(* CODESYS project TcDynCollections.library
   Company: FisoThemes
   DefaultNamespace: TcDynCollections
   Version: 0.3.1.0
   DocFormat: reStructuredText
   Placeholder: TwinCat Dynamic Collections
   Author: Goodwill Mzumala
   Description: A library for handling collections of data dynamically.
   Title: TwinCat Dynamic Collections

Project tree, tasks and I/O mapping:
  libraries: Tc2_Standard, * (Beckhoff Automation GmbH); Tc2_System, * (Beckhoff Automation GmbH); Tc2_Utilities, 3.3.38.0 (Beckhoff Automation GmbH); Tc3_Module, * (Beckhoff Automation GmbH)
  DUTs/
    Aliases/
      data type T_BST_Node
      data type T_BST_Traversal
      data type T_Capacity
      data type T_Error
      data type T_Generic
      data type T_Generic_Ex
      data type T_Hash_Code
      data type T_Query_Interface
      data type T_Type
    Enums/
      data type E_BINARY_SEARCH_TREE_TRAVERSAL
    Interfaces/
      interface I_Binary_Search_Tree: _Type, Balance, Find, Insert, Remove, Traverse
      interface I_Collection: _Count, _Error_Status, _Is_Empty, Clear
      interface I_Deque: Back, Dequeue_At_Back, Dequeue_At_Front, Dequeue_Void_At_Back, Dequeue_Void_At_Front, Enqueue_At_Back, Enqueue_At_Front, Front, Peek, Reverse
      interface I_Generic_Binary_Search_Tree: Find_Generic, Insert_Generic
      interface I_Generic_Collection
      interface I_Generic_List: Get_Generic, Insert_Generic
      interface I_List: Add_Back, Add_Front, Contains, Find, Get, Get_First, Get_Last, Get_Value_As_String, Insert, Remove, Remove_At, Remove_Last, Resize, Reverse, Set
      interface I_Map: _Keys, _Values, Get, Insert, Remove, Update
      interface I_Queue: Dequeue, Dequeue_Void, Enqueue, Enqueue_At_Front, Peek, Reverse
      interface I_Read_Only_List: Clear, Contains, Find, Get, Get_First, Get_Last, Get_Value_As_String
      interface I_Stack: Peek, Pop, Pop_Void, Push, Reverse, Top
      interface I_Tree_Map: _Traversal, Balance
      interface I_Write_Only_List: _Count, _Is_Empty, Add_Back, Add_Front, Clear, Insert, Remove, Remove_At, Remove_Last, Resize, Reverse, Set
    Structs/
      data type ST_BINARY_SEARCH_TREE_NODE
      data type ST_ERROR
      data type ST_GENERIC
      data type ST_HASH_MAP_ENTRY
      data type ST_LIST_NODE
      data type ST_TREE_MAP_ENTRY_NODE
  GVLs/
    global variables GVL_CmpErrors
  POUs/
    Examples/
      program P_Example_Array_List [ST]: Scrub
      program P_Example_Binary_Search_Tree [ST]
      program P_Example_List [ST]: Scrub
      program P_Example_Queue [ST]
      program P_Example_Stack [ST]
      program P_Example_Tree_Map [ST]: Scrub
    Function Blocks/
      Helpers/
        function block FB_Helper_BST_Balancer [ST]
        function block FB_Helper_Tree_Map_Balancer [ST]
      function block FB_Array_List [ST]: EmptyListException, LessThanZeroException, MemCmpErrExpection, OutOfBoundsException, TypeMismatchException, CopyValueTo, DecrementCount, Free_Value, GetValueAsString, IncrementCount, Internal_Add_Back, Internal_Add_Front, Internal_Set, Malloc_Array, Malloc_Value, SetValue, _Is_Empty, Add_Back, Add_Front, Clear, Contains, FB_exit, FB_init, Find, Get, Get_First, Get_Generic, Get_Last, Get_Value_As_String, Insert, Insert_Generic, Remove, Remove_At, Remove_Last, Resize, Reverse, Set
      function block FB_Binary_Search_Tree [ST]: InvalidTypeException, Balance_Ready, Compare, Internal_Find, Internal_Insert, Internal_Remove, Is_Balanced, Malloc_Node, _Type, Balance, Clear, FB_exit, FB_init, Find, Find_Generic, Insert, Insert_Generic, Remove, Traverse
      function block FB_Collection [ST]: ClearException, EmptyListException, FailedInsertionException, NullReferenceException, OutOfBoundsException, RaiseException, ValueFoundException, ValueNotFoundException, ClearValue, CopyValueTo, DecrementCount, IncrementCount, _Count, _Error_Status, _Is_Empty, Clear
      function block FB_Hash_Map [ST]: Populate_Bucket_List, FB_init, Get, Insert, Remove, Remove_Void, Update
      function block FB_List [ST]: EmptyListException, MemCmpErrExpection, OutOfBoundsException, TypeMismatchException, CopyValueTo, DecrementCount, Free_Node, GetValueAsString, IncrementCount, Iterate, Malloc_Node, SetValue, _Is_Empty, Add_Back, Add_Front, Clear, Contains, FB_exit, FB_init, Find, Get, Get_First, Get_Generic, Get_Last, Get_Value_As_String, Insert, Insert_Generic, Remove, Remove_At, Remove_Last, Resize, Reverse, Set
      function block FB_Queue [ST]: NullReferenceException, _Count, _Error_Status, _Is_Empty, CatchError, Clear, Dequeue, Dequeue_Void, Enqueue, Enqueue_At_Front, Peek, Reverse
      function block FB_Read_Only_List [ST]: NullReferenceException, _Count, _Error_Status, _Is_Empty, Clear, Contains, Find, Get, Get_First, Get_Last, Get_Value_As_String
      function block FB_Stack [ST]: NullReferenceException, CatchError, _Count, _Error_Status, _Is_Empty, Clear, Peek, Pop, Pop_Void, Push, Reverse, Top
      function block FB_Tree_Map [ST]: Balance_Ready, Compare, Copy_Value, Internal_Get, Internal_Insert, Internal_Remove, Internal_Traversal, Internal_Update, Malloc_Node, Malloc_Value, _Keys, _Traversal, _Values, Balance, Clear, FB_exit, Get, Insert, Remove, Update
      function block FB_Write_Only_List [ST]: NullReferenceException, _Count, _Error_Status, _Is_Empty, Add_Back, Add_Front, Clear, Insert, Remove, Remove_At, Remove_Last, Resize, Reverse, Set
    Functions/
      function F_Error [ST]
    program MAIN [ST]
  Project Information/
    function F_GetCompany [ST]
    function F_GetTitle [ST]
    function F_GetVersion [ST]
  UML/
    Array List UML
    List UML
    Queue UML
    Stack UML
    TwinCAT Dynamic Collections Interface UML
  Version/
    global variables Global_Version
  VISUs/
*)

// DUTs/Aliases/T_BST_Node
TYPE T_BST_Node : ST_BINARY_SEARCH_TREE_NODE; END_TYPE

// DUTs/Aliases/T_BST_Traversal
TYPE T_BST_Traversal : E_BINARY_SEARCH_TREE_TRAVERSAL; END_TYPE

// DUTs/Aliases/T_Capacity
TYPE T_Capacity : DINT; END_TYPE

// DUTs/Aliases/T_Error
TYPE T_Error : ST_ERROR; END_TYPE

// DUTs/Aliases/T_Generic
// Type ANY
TYPE T_Generic : __SYSTEM.AnyType; END_TYPE

// DUTs/Aliases/T_Generic_Ex
// Type ANY in struct format extended with value of type STRING(255)
TYPE T_Generic_Ex : ST_GENERIC; END_TYPE

// DUTs/Aliases/T_Hash_Code
TYPE T_Hash_Code : LWORD; END_TYPE

// DUTs/Aliases/T_Query_Interface
TYPE T_Query_Interface : __SYSTEM.IQueryInterface; END_TYPE

// DUTs/Aliases/T_Type
TYPE T_Type : __SYSTEM.TYPE_CLASS; END_TYPE

// DUTs/Enums/E_BINARY_SEARCH_TREE_TRAVERSAL
{attribute 'qualified_only'}
{attribute 'strict'}
TYPE E_BINARY_SEARCH_TREE_TRAVERSAL :
(
	Inorder := 0,
	Preorder,
	Postorder, 
	Level_Order
)BYTE;
END_TYPE

// DUTs/Structs/ST_BINARY_SEARCH_TREE_NODE
(* Node for Binary Search Tree *)
{attribute 'enable_dynamic_creation'}
TYPE INTERNAL ST_BINARY_SEARCH_TREE_NODE :
STRUCT
	Data 		: T_Generic;
	pLeft 		: POINTER TO ST_BINARY_SEARCH_TREE_NODE;
	pRight 		: POINTER TO ST_BINARY_SEARCH_TREE_NODE;
END_STRUCT
END_TYPE

// DUTs/Structs/ST_ERROR
(* STRUCT used to contain error status information. *)
{attribute 'enable_dynamic_creation'}
TYPE ST_ERROR :
STRUCT
	bSTATUS : BOOL; 		// Indicates if an error has occurred | TRUE = error, FALSE = no error
	nCODE 	: DINT; 		// Error code specific to the particular error.
	sSOURCE : T_MaxString; 	// Textual information describing the error.
END_STRUCT
END_TYPE

// DUTs/Structs/ST_GENERIC
(* Generic data type used for Programs/Functions/Function Blocks to handle data in a generic way. *)
{attribute 'enable_dynamic_creation'}
TYPE ST_GENERIC EXTENDS __SYSTEM.AnyType :
STRUCT
	sValue 	: T_MaxString; 	// Data of parameter as a string for easy convertion.
END_STRUCT
END_TYPE

// DUTs/Structs/ST_HASH_MAP_ENTRY
// Entry for a map in the form of a key-value pair
{attribute 'enable_dynamic_creation'}
TYPE INTERNAL ST_HASH_MAP_ENTRY :
STRUCT
	Hash_Code 		: T_Hash_Code; 	// Hash code of key
	Key 			: T_Generic_Ex; 	// Key used to identify stored value
	Value 			: T_Generic_Ex; 	// Value to store in dictionary with key
END_STRUCT
END_TYPE

// DUTs/Structs/ST_LIST_NODE
(* Node for linked list*)
{attribute 'enable_dynamic_creation'}
TYPE INTERNAL ST_LIST_NODE:
STRUCT
	Data 		: T_Generic_Ex; // Stored data.
	pPrevious 	: POINTER TO ST_LIST_NODE := Tc3_Module.GVL.NULL; 	// Pointer to previous node.
	pNext 		: POINTER TO ST_LIST_NODE := Tc3_Module.GVL.NULL; 	// Pointer to next node.
END_STRUCT
END_TYPE

// DUTs/Structs/ST_TREE_MAP_ENTRY_NODE
// Node for a tree map
{attribute 'enable_dynamic_creation'}
TYPE INTERNAL ST_TREE_MAP_ENTRY_NODE :
STRUCT
	Key 	: T_Generic; 					// Key used to identify stored value
	Value 	: T_Generic; 					// Value to store in dictionary with key
	pLeft 	: POINTER TO ST_TREE_MAP_ENTRY_NODE;
	pRight 	: POINTER TO ST_TREE_MAP_ENTRY_NODE;
END_STRUCT
END_TYPE

// GVLs/GVL_CmpErrors
{attribute 'qualified_only'}
(* Error code are @ CmpErrors.Errors.<variable> from the CmpErrors2 Interfaces library.*)
VAR_GLOBAL CONSTANT
	ERR_OK 						: DINT	:= 16#0;  	//	Ok
	ERR_FAILED 					: DINT	:= 16#1;  	//	General error - To be used only for INTERNAL errors
	ERR_PARAMETER 				: DINT	:= 16#2;  	//	Invalid parameter for this operation
	ERR_NOTINITIALIZED 			: DINT	:= 16#3;  	//	Function cannot be executed, since component has not been initialized yet. It may work later, though
	ERR_VERSION 				: DINT	:= 16#4;  	//	Version conflict
	ERR_TIMEOUT 				: DINT	:= 16#5;  	//	Operation timed out
	ERR_NOBUFFER 				: DINT	:= 16#6;  	//	Insufficient memory to carry out the request
	ERR_PENDING 				: DINT	:= 16#A;  	//	FOR async-calls: call not complete, yet
	ERR_NUMPENDING 				: DINT	:= 16#B;  	//  TO many pending calls. Try later
	ERR_NOTIMPLEMENTED 			: DINT	:= 16#C;  	//  The function is not implemented
	ERR_INVALIDID 				: DINT	:= 16#D;  	//  No object with the provided id found
	ERR_OVERFLOW 				: DINT	:= 16#E;  	//	Integer overflow
	ERR_BUFFERSIZE 				: DINT	:= 16#F;  	//	The size of a buffer is too small OR invalid
	ERR_NO_OBJECT 				: DINT	:= 16#10;  	//	No object with THIS specified name available
	ERR_NOMEMORY 				: DINT	:= 16#11;  	//  No heap memory available
	ERR_DUPLICATE 				: DINT	:= 16#12A;  //  n object with the same name is still available
	ERR_MEMORY_OVERWRITE 		: DINT	:= 16#13;  	//  Heap memory was written out of bounds! Memory overwrite error
	ERR_INVALID_HANDLE 			: DINT	:= 16#14;  	//  Invalid handle to an object
	ERR_END_OF_0BJECT 			: DINT := 16#15;  	//  End OF object reached
	ERR_NO_CHANGE 				: DINT := 16#16;  	//  No changes done
	ERR_INVALID_INTERFACE 		: DINT := 16#17;  	//  Invalid OR unknown INTERFACE
	ERR_NOT_SUPPORTED 			: DINT := 16#18;  	//  Functionality not supported
	ERR_NO_ACCESS_RIGHTS 		: DINT := 16#19;  	//  No access rights for this operation
	ERR_OUT_OF_LIMITS 			: DINT := 16#1A;  	//  Specified limits of a resource exceeded
	ERR_ENTRIES_REMAINING 		: DINT := 16#18;  	//  Remaining entries that could not be transmitted because of buffer limitation
	ERR_INVALID_SESSION_ID 		: DINT := 16#1C;  	//  Invalid online sessionid
	ERR_EXCEPTION 				: DINT := 16#1D;  	//  Exception occurred
	ERR_SIGNATURE_MISMATCH 		: DINT := 16#1E;	//	Signature mismatch OF an api function
	ERR_VERSION_MISMATCH 		: DINT := 16#1F;	//	Version mismatch
	ERR_TYPE_MISMATCH 			: DINT := 16#20;	//	TYPE mismatch
	ERR_ID_MISMATCH 			: DINT := 16#21;	//	ID mismatch
	ERR_NO_CONSISTENCY 			: DINT := 16#22;	//	Consistency error
	ERR_NO_COMM_CYCLE 			: DINT := 16#23;	//	No COMM_CYCLE needed
	ERR_DONT_SUSPEND_TASK 		: DINT := 16#24;	//	DO NOT suspend task after an exception
	ERR_MEMORY_LOCK_FAILED 		: DINT := 16#25;	//	Memory cannot be locked in THIS operation
	ERR_LICENSE_MISSING 		: DINT := 16#26;	//	License missing FOR the runtime
	ERR_OPERATION_DENIED 		: DINT := 16#27;	//	Operation denied 
	ERR_DEVICE 					: DINT := 16#28;	//	Device error
	ERR_DISK_FULL 				: DINT := 16#29;	//	Disk full
	ERR_CRC_FAILED 				: DINT := 16#30;	//	INTERNAL use in runtime
	ERR_MEDIA_ERASE 			: DINT := 16#31;	//	INTERNAL use in runtime
	ERR_FILE_ERROR 				: DINT := 16#32;	//	File error. e.g. cannot open a file for writing because it could be write PROTECTED
	ERR_NO_RETAIN_MEMORY 		: DINT := 16#33;	//	No RETAIN memory available
	ERR_OUT_OF_LIMITS_MIN 		: DINT := 16#34;	//	Specified minimum-limit of a resource exceeded
	ERR_OUT_OF_LIMITS_MAX 		: DINT := 16#35;	//	Specified maximum-limit of a resource exceeded
	ERR_SIZE_MISMATCH 			: DINT := 16#36;	//	Size mismatch
	ERR_CALL_AGAIN 				: DINT := 16#37;	//	Operation is not yet finished, call FUNCTION again to proceed
	ERR_NOTHING_TO_DO 			: DINT := 16#38;	//	Operation has nothing to do. No execution.
	ERR_SECURITY_CHECKS_FAILED 	: DINT := 16#39;	//	Some security checks have failed. /* This is a generic error code to report this error over public channels. In this case the error code doesn’t provide a detailed cause for the error. */
	ERR_INVALID_SEQUENCE 		: DINT := 16#3A;	//	 
	ERR_INVALID_REFERENCE 		: DINT := 16#3B;	//	Dereferencing an IEC reference in IecVarAccess failed due TO invalid destination address, e. G. NULL.
	ERR_CONVERSION_INCOMPLETE 	: DINT := 16#3C;	//	Conversion OF STRING encodings was NOT lossless.
	ERR_SOCK_NOTINITIALIZED 	: DINT := 16#201;   //  Socket errors (range: 0x0200 - 0X02FF)
	ERR_SOCK_NOTSOCKET 			: DINT := 16#202;   //  The provided socket handle is invalid
	ERR_SOCK_AFUNSUPPORTED 		: DINT := 16#203;   //  The address family is NOT supported
	ERR_SOCK_PROTOUNSUPPORTED  	: DINT := 16#204;   //  Protocol is NOT supported */
	ERR_SOCK_NOBUFFER 			: DINT := 16#205;   //  NOT enough buffer TO handle the request */
	ERR_SOCK_WOULDBLOCK 		: DINT := 167206;   //  Socket is in nonblocking mode but THIS call would block =/
	ERR_SOCK_ADDRINUSE 			: DINT := 16#207;   //  The provided address is already in use */
	ERR_SOCK_ADDRNOTAVAILABLE  	: DINT := 16#208;   //  The provided address is NOT available on THIS computer */
	ERR_SOCK_CONNREFUSED 		: DINT := 16#209;   //  Connection has been refused BY the remote host */
	ERR_SOCK_TIMEDOUT 			: DINT := 16#20A;   //  Operation timed out */
	ERR_SOCK_HOSTNOTFOUND 		: DINT := 16#208;   //  The host has NOT been found */
	ERR_SOCK_HOSTUNREACHABLE  	: DINT := 16#20C;   //  Host is unreachable */
	ERR_SOCK_1SCONNECTED 		: DINT := 16#20D;   //  Socket is already connected =/
	ERR_SOCK_NOTCONNECTED 		: DINT := 16#20E;   //  The socket is NOT connected */
	ERR_SOCK_SHUTDOWN 			: DINT := 16#20F;   //  Shutdown has been called on the socket =/
	ERR_SOCK_MSGSIZE 			: DINT := 16#210;   //  FOR sockets OF TYPE DGRAM. The package TO send exceeds the maximum package size =/
	ERR_SOCK_CLOSED 			: DINT := 167211;   //  Socket has been gracefully closed. No more send/receives allowed =/
	ERR_L7_TAG_MISSING 			: DINT := 16#300;	//  Tag missing in online communication buffer
	ERR_L7_UNKNOWNCMDGROUP 		: DINT := 16#301;	//  Unknown command group
	ERR_L7_UNKNOWNCMD 			: DINT := 16#302;	//  Unknown command (within a valid command group)
	ERR_L7_INCOMPLETE 			: DINT := 16#303;	//  Level 7 service incomplete
END_VAR

// Version/Global_Version
{attribute 'TcGenerated'}
{attribute 'no-analysis'}
{attribute 'linkalways'}
// This function has been automatically generated from the project information.
VAR_GLOBAL CONSTANT
	{attribute 'const_non_replaced'}
	stLibVersion_TwinCat_Dynamic_Collections : ST_LibVersion := (iMajor := 0, iMinor := 3, iBuild := 1, iRevision := 0, nFlags := 0, sVersion := '0.3.1.0');
END_VAR

// DUTs/Interfaces/I_Binary_Search_Tree
// Interface for binary search tree
INTERFACE I_Binary_Search_Tree EXTENDS I_Collection

// Gets the type of the data on the binary search tree
PROPERTY _Type : T_Type
GET
END_GET
END_PROPERTY

// Balances Binary Search Tree. Tree will normal auto balance every time its count is a multiple of 4
METHOD Balance
END_METHOD

(* Checks if data is contained in binary search tree *)
METHOD Find : I_Binary_Search_Tree
VAR_INPUT
	Data 	: ANY; 	// Data to remove
END_VAR
VAR_OUTPUT
	bFound 	: BOOL; 		// Indicates whether data was found. Found = TRUE, Not Found = FALSE
END_VAR
END_METHOD

(* Insert data into binary search tree *)
METHOD Insert 	: I_Binary_Search_Tree
VAR_INPUT
	Data 		: ANY; // Data to insert
END_VAR
VAR_OUTPUT
	bSuccess 	: BOOL; // Indicates whether operation was successful. Success = TRUE, Failure = FALSE
END_VAR
END_METHOD

(* Removes data from binary search tree *)
METHOD Remove : I_Binary_Search_Tree
VAR_INPUT
	Data 		: ANY; // Data to remove
END_VAR
VAR_OUTPUT
	bSuccess 	: BOOL; // Indicates whether operation was successful. Success = TRUE, Failure = FALSE
END_VAR
END_METHOD

(* Traveses the binary search tree and appends into a collection *)
METHOD Traverse : I_Binary_Search_Tree
VAR_INPUT
	eMethod 		: T_BST_Traversal; // Method to traverse the binary search tree
	ipGeneric_List 	: I_Generic_List; 		// Collection to append data to.
END_VAR
END_METHOD

END_INTERFACE

// DUTs/Interfaces/I_Collection
INTERFACE I_Collection EXTENDS __SYSTEM.IQueryInterface

// Number of items in the collection
PROPERTY _Count : T_Capacity
GET
END_GET
END_PROPERTY

(* Gets Function Block's error status *)
PROPERTY _Error_Status : T_Error
GET
END_GET
END_PROPERTY

// Checks if collection is empty
PROPERTY _Is_Empty : BOOL
GET
END_GET
END_PROPERTY

// Empties/Clears/Deletes every item in the collection
METHOD Clear
END_METHOD

END_INTERFACE

// DUTs/Interfaces/I_Generic_List
// Interface operating with generic data contained in a list.
INTERFACE I_Generic_List EXTENDS I_Generic_Collection

// Gets a value from a list in it's generic form.
// (* Use carefully as this contains the pointer of the actual value in the collection. *)
// If you wish to use this it is recommeded you create a copy of the returned value using MEMMOVE or MEMCPY
METHOD Get_Generic : I_Generic_List
VAR_INPUT
	nIndex 		: T_Capacity; 			// Location of item
END_VAR
VAR_OUTPUT
	Return_Item : T_Generic;  	// Variable to store returned item
	bSuccess 	: BOOL;
END_VAR
END_METHOD

// Adds new item to list at specified location using the generic form. 
// If index = 0, item will be added at the front, if index = count, item will be added at the back
METHOD Insert_Generic : I_Generic_List
VAR_INPUT
	Item 	 : T_Generic;  	// Item to store in list
	nIndex 	 : T_Capacity; 			// Location of item
END_VAR
VAR_OUTPUT
	bSuccess : BOOL;
END_VAR
END_METHOD

END_INTERFACE

// DUTs/Interfaces/I_Generic_Collection
// Interface handling generic data contained in a collection.
INTERFACE I_Generic_Collection EXTENDS I_Collection

END_INTERFACE

// DUTs/Interfaces/I_Deque
// Interface for a ouble ended queue - Dequeu
INTERFACE I_Deque EXTENDS I_Collection

(* Get item at the back of the deque without removing it. *)
METHOD Back : I_Deque
VAR_INPUT
	Item 	: ANY; (* Variable to store returned item value *)
END_VAR
VAR_OUTPUT
	bSuccess : BOOL;
END_VAR
END_METHOD

(* Gets and remove item at the front of the deque *)
METHOD Dequeue_At_Back : I_Deque
VAR_INPUT
	Item : ANY; (* Variable to store returned item value *)
END_VAR
VAR_OUTPUT
	bSuccess : BOOL;
END_VAR
END_METHOD

(* Gets and remove item at the front of the deque *)
METHOD Dequeue_At_Front : I_Deque
VAR_INPUT
	Item : ANY; (* Variable to store returned item value *)
END_VAR
VAR_OUTPUT
	bSuccess : BOOL;
END_VAR
END_METHOD

(* Removes item at the back of the deque without returning anything *)
METHOD Dequeue_Void_At_Back : I_Deque
VAR_OUTPUT
	bSuccess : BOOL;
END_VAR
END_METHOD

(* Removes item at the front of the deque without returning anything *)
METHOD Dequeue_Void_At_Front : I_Deque
VAR_OUTPUT
	bSuccess : BOOL;
END_VAR
END_METHOD

(* Adds item at the back of the deque *)
METHOD Enqueue_At_Back : I_Deque
VAR_INPUT
	Item : ANY; (* Variable containg data to store on the queue *)
END_VAR
VAR_OUTPUT
	bSuccess : BOOL;
END_VAR
END_METHOD

(* Adds item at the front of the deque *)
METHOD Enqueue_At_Front : I_Deque
VAR_INPUT
	Item : ANY; (* Variable containg data to store on the queue *)
END_VAR
VAR_OUTPUT
	bSuccess : BOOL;
END_VAR
END_METHOD

(* Get item at the front of the deque without removing it. *)
METHOD Front : I_Deque
VAR_INPUT
	Item 	: ANY; (* Variable to store returned item value *)
END_VAR
VAR_OUTPUT
	bSuccess : BOOL;
END_VAR
END_METHOD

(* Get item from the deque without removing it. *)
METHOD Peek : I_Deque
VAR_INPUT
	Item 	: ANY; (* Variable to store returned item value *)
	nIndex 	: DINT; (* Location of item*)
END_VAR
VAR_OUTPUT
	bSuccess : BOOL;
END_VAR
END_METHOD

(* Reverses the order of items in the deque *)
METHOD Reverse : I_Deque
VAR_OUTPUT
	bSuccess : BOOL;
END_VAR
END_METHOD

END_INTERFACE

// DUTs/Interfaces/I_Generic_Binary_Search_Tree
// Interface operating with generic data contained in a list.
INTERFACE I_Generic_Binary_Search_Tree EXTENDS I_Generic_Collection

// Checks if generic data is inside binary search tree
METHOD Find_Generic : I_Generic_Binary_Search_Tree
VAR_INPUT
	Data 		: T_Generic; 	// Generic Data to find
END_VAR
VAR_OUTPUT
	bFound 		: BOOL; // Indicates whether data was found. Found = TRUE, Not Found = FALSE
END_VAR
END_METHOD

// Adds new generic item at into binary search tree.
// The binary seach tree will store a copy of the generic item so as to not modify the original value outside it's scope.
METHOD Insert_Generic : I_Generic_Binary_Search_Tree
VAR_INPUT
	Data 	: T_Generic; // Item to store
END_VAR
VAR_OUTPUT
	bSuccess 	: BOOL; // Indicates whether operation was successful. Success = TRUE, Failure = FALSE
END_VAR
END_METHOD

END_INTERFACE

// DUTs/Interfaces/I_List
INTERFACE I_List EXTENDS I_Collection

// Adds an item to the end of the list
METHOD Add_Back : I_List
VAR_INPUT
	Item 	: ANY; // Value to store in list
END_VAR
VAR_OUTPUT
	bSuccess : BOOL;
END_VAR
END_METHOD

// Adds an item at the front of the list
METHOD Add_Front : I_List
VAR_INPUT
	Item 	: ANY; // Value to store in list
END_VAR
VAR_OUTPUT
	bSuccess : BOOL;
END_VAR
END_METHOD

(* Checks if item is contained in list *)
METHOD Contains : BOOL
VAR_INPUT
	Item : ANY; // Item to find in list
END_VAR
END_METHOD

// Find the location of an item in list.
METHOD Find : I_List
VAR_INPUT
	Item 	: ANY; // Item to find in list
END_VAR
VAR_OUTPUT
	nIndex	 : T_Capacity; //Location of item in list 
	bSuccess : BOOL;
END_VAR
END_METHOD

// Gets item from list at specified location without removing it
METHOD Get : I_List
VAR_INPUT
	Return_Item 	: ANY;  // Variable to store returned item
	nIndex 			: T_Capacity; // Location of item
END_VAR
VAR_OUTPUT
	bSuccess : BOOL;
END_VAR
END_METHOD

// Gets item at the front of the list 
METHOD Get_First : I_List
VAR_INPUT
	Return_Item 	: ANY; // Variable to store returned item
END_VAR
VAR_OUTPUT
	bSuccess : BOOL;
END_VAR
END_METHOD

// Gets item at the back of the list 
METHOD Get_Last : I_List
VAR_INPUT
	Return_Item 	: ANY; // Variable to store returned item
END_VAR
VAR_OUTPUT
	bSuccess : BOOL;
END_VAR
END_METHOD

// Returns item as a string, if type to string conversion is supported
METHOD Get_Value_As_String : I_List
VAR_INPUT
	nIndex	: T_Capacity; // Location of item
END_VAR
VAR_OUTPUT
	sItem 	: T_MaxString; // Variable to store returned item
END_VAR
END_METHOD

// Adds new item to list at specified location, if index = 0, item will be added at the front, if index = count, item will be added at the back
METHOD Insert : I_List
VAR_INPUT
	Item 	: ANY;  // Item to store in list
	nIndex 	: T_Capacity; // Location of item
END_VAR
VAR_OUTPUT
	bSuccess : BOOL;
END_VAR
END_METHOD

// Removes item at the front of the list and returns nothing
METHOD Remove : I_List
VAR_OUTPUT
	bSuccess : BOOL;
END_VAR
END_METHOD

// Remove item at specified location and return nothing
METHOD Remove_At : I_List
VAR_INPUT
	nIndex : T_Capacity; // Location of item
END_VAR
VAR_OUTPUT
	bSuccess : BOOL;
END_VAR
END_METHOD

// Removes item at the back of the list and returns nothing
METHOD Remove_Last : I_List
VAR_OUTPUT
	bSuccess : BOOL;
END_VAR
END_METHOD

// Manually resize list. If list becomes smaller, item on higher locations will be deleted.
METHOD Resize : I_List
VAR_INPUT
	nSize : T_Capacity; // New size of list.
END_VAR
VAR_OUTPUT
	bSuccess : BOOL;
END_VAR
END_METHOD

// Reverses the order of items in the list
METHOD Reverse : I_List
VAR_OUTPUT
	bSuccess : BOOL;
END_VAR
END_METHOD

// Adds new item to list in the specified location without resizing list
METHOD Set : I_List
VAR_INPUT
	Item 	: ANY; 	// Item to store in list
	nIndex 	: T_Capacity; // Location of item
END_VAR
VAR_OUTPUT
	bSuccess : BOOL;
END_VAR
END_METHOD

END_INTERFACE

// DUTs/Interfaces/I_Map
// An interface for a collection that holds key/value pairs  
INTERFACE I_Map EXTENDS I_Collection

// Gets a read-only list of the keys
PROPERTY _Keys : I_Read_Only_List
GET
END_GET
END_PROPERTY

// Gets a read-only list of the values
PROPERTY _Values : I_Read_Only_List
GET
END_GET
END_PROPERTY

// Gets the value associated with the specified key without remocing it from the dictionary
METHOD Get : I_Map
VAR_INPUT
	Key 			: ANY; // Key used to identify stored value
	Return_Value 	: ANY; // Variable to store requested data 
END_VAR
VAR_OUTPUT
	bSuccess : BOOL;
END_VAR
END_METHOD

// Insert an element with the provided key and value to the map
METHOD Insert : I_Map
VAR_INPUT
	Key 	: ANY; // Key used to identify stored value
	Value 	: ANY; // Value to store in map with key
END_VAR
VAR_OUTPUT
	bSuccess : BOOL;
END_VAR
END_METHOD

// Removes value with the specified key from the map
METHOD Remove : I_Map
VAR_INPUT
	Key : ANY; // Key used to identify stored value
END_VAR
VAR_OUTPUT
	bSuccess : BOOL;
END_VAR
END_METHOD

// Updates the value an element with the provided key and value in the map
METHOD Update : I_Map
VAR_INPUT
	Key 	: ANY; // Key used to identify stored value
	Value 	: ANY; // Value to store in map with key
END_VAR
VAR_OUTPUT
	bSuccess : BOOL;
END_VAR
END_METHOD

END_INTERFACE

// DUTs/Interfaces/I_Read_Only_List
// Implement this with I_List to allow a list to be ready only. 
INTERFACE I_Read_Only_List EXTENDS I_Collection

(* DOES NOTHING *)
METHOD Clear
END_METHOD

(* Checks if item is contained in list *)
METHOD Contains : BOOL
VAR_INPUT
	Item : ANY; // Item to find in list
END_VAR
END_METHOD

// Find the location of an item in list.
METHOD Find : I_Read_Only_List
VAR_INPUT
	Item 	: ANY; // Item to find in list
END_VAR
VAR_OUTPUT
	nIndex	: DINT; //Location of item in list 
	bSuccess : BOOL;
END_VAR
END_METHOD

// Gets item from list at specified location without removing it
METHOD Get : I_Read_Only_List
VAR_INPUT
	Return_Item 	: ANY;  // Variable to store returned item
	nIndex 			: DINT; // Location of item
END_VAR
VAR_OUTPUT
	bSuccess : BOOL;
END_VAR
END_METHOD

// Gets item at the front of the list 
METHOD Get_First : I_Read_Only_List
VAR_INPUT
	Return_Item 	: ANY; // Variable to store returned item
END_VAR
VAR_OUTPUT
	bSuccess : BOOL;
END_VAR
END_METHOD

// Gets item at the back of the list 
METHOD Get_Last : I_Read_Only_List
VAR_INPUT
	Return_Item 	: ANY; // Variable to store returned item
END_VAR
VAR_OUTPUT
	bSuccess : BOOL;
END_VAR
END_METHOD

// Returns item as a string, if type to string conversion is supported
METHOD Get_Value_As_String : I_Read_Only_List
VAR_INPUT
	nIndex	: DINT; // Location of item
END_VAR
VAR_OUTPUT
	sItem 	: T_MaxString; // Variable to store returned item
END_VAR
END_METHOD

END_INTERFACE

// DUTs/Interfaces/I_Queue
INTERFACE I_Queue EXTENDS I_Collection

(* Gets and remove item at the front of the queue *)
METHOD Dequeue : I_Queue
VAR_INPUT
	Item : ANY; (* Variable to store returned item value *)
END_VAR
VAR_OUTPUT
	bSuccess : BOOL;
END_VAR
END_METHOD

(* Removes item at the front of the queue without returning anything *)
METHOD Dequeue_Void : I_Queue
VAR_OUTPUT
	bSuccess : BOOL;
END_VAR
END_METHOD

(* Adds item at the back of the queue *)
METHOD Enqueue : I_Queue
VAR_INPUT
	Item : ANY; (* Variable containg data to store on the queue *)
END_VAR
VAR_OUTPUT
	bSuccess : BOOL;
END_VAR
END_METHOD

(* Adds item at the front of the queue *)
METHOD Enqueue_At_Front : I_Queue
VAR_INPUT
	Item : ANY; (* Variable containg data to store on the queue *)
END_VAR
VAR_OUTPUT
	bSuccess : BOOL;
END_VAR
END_METHOD

(* Get item from the queue without removing it. *)
METHOD Peek : I_Queue
VAR_INPUT
	Item 	: ANY; (* Variable to store returned item value *)
	nIndex 	: DINT; (* Location of item*)
END_VAR
VAR_OUTPUT
	bSuccess : BOOL;
END_VAR
END_METHOD

METHOD Reverse : I_Queue
VAR_OUTPUT
	bSuccess : BOOL;
END_VAR
END_METHOD

END_INTERFACE

// DUTs/Interfaces/I_Stack
INTERFACE I_Stack EXTENDS I_Collection

(* Get item from stack without removing it. *)
METHOD Peek : I_Stack
VAR_INPUT
	Item 	 : ANY; (* Variable to store returned item value *)
	nIndex 	 : DINT; (* Location of item*)
END_VAR
VAR_OUTPUT
	bSuccess : BOOL;
END_VAR
END_METHOD

(* Gets and deletes item at the top of the stack *)
METHOD Pop : I_Stack
VAR_INPUT
	Item : ANY; (* Variable to store returned item value *)
END_VAR
VAR_OUTPUT
	bSuccess : BOOL;
END_VAR
END_METHOD

(* Removes item at the top of the stack without returning anything *)
METHOD Pop_Void : I_Stack
VAR_OUTPUT
	bSuccess : BOOL;
END_VAR
END_METHOD

(* Add item to the top of the stack *)
METHOD Push : I_Stack
VAR_INPUT
	Item : ANY; (* Variable containg data to store on the stack *)
END_VAR
VAR_OUTPUT
	bSuccess : BOOL;
END_VAR
END_METHOD

(* Reverses order of items on stack *)
METHOD Reverse : I_Stack
VAR_OUTPUT
	bSuccess : BOOL;
END_VAR
END_METHOD

(* Get item at the top of the stack without removing it. *)
METHOD Top : I_Stack
VAR_INPUT
	Item 	: ANY; (* Variable to store returned item value *)
END_VAR
VAR_OUTPUT
	bSuccess : BOOL;
END_VAR
END_METHOD

END_INTERFACE

// DUTs/Interfaces/I_Tree_Map
// An interface for a collection that holds key/value pairs  
INTERFACE I_Tree_Map EXTENDS I_Map

// Get and set the order in which the property _Keys/Value should return values
PROPERTY _Traversal : T_BST_Traversal
GET
END_GET
SET
END_SET
END_PROPERTY

// Balances Tree Map. Tree will normal auto balance every time its count is a multiple of 4
METHOD Balance
END_METHOD

END_INTERFACE

// DUTs/Interfaces/I_Write_Only_List
INTERFACE I_Write_Only_List EXTENDS I_Collection

(* Returns -1, this is a write-only list*)
PROPERTY _Count : DINT
GET
END_GET
END_PROPERTY

(* Returns FALSE as this is a write-only list *)
PROPERTY _Is_Empty : BOOL
GET
END_GET
END_PROPERTY

// Adds an item to the end of the list
METHOD Add_Back : I_Write_Only_List
VAR_INPUT
	Item 	: ANY; // Value to store in list
END_VAR
VAR_OUTPUT
	bSuccess : BOOL;
END_VAR
END_METHOD

// Adds an item at the front of the list
METHOD Add_Front : I_Write_Only_List
VAR_INPUT
	Item 	: ANY; // Value to store in list
END_VAR
VAR_OUTPUT
	bSuccess : BOOL;
END_VAR
END_METHOD

// Empties/Clears/Deletes every item in the collection
METHOD Clear
END_METHOD

// Adds new item to list at specified location, if index = 0, item will be added at the front, if index = count, item will be added at the back
METHOD Insert : I_Write_Only_List
VAR_INPUT
	Item 	: ANY;  // Item to store in list
	nIndex 	: DINT; // Location of item
END_VAR
VAR_OUTPUT
	bSuccess : BOOL;
END_VAR
END_METHOD

// Removes item at the front of the list and returns nothing
METHOD Remove : I_Write_Only_List
VAR_OUTPUT
	bSuccess : BOOL;
END_VAR
END_METHOD

// Remove item at specified location and return nothing
METHOD Remove_At : I_Write_Only_List
VAR_INPUT
	nIndex : DINT; // Location of item
END_VAR
VAR_OUTPUT
	bSuccess : BOOL;
END_VAR
END_METHOD

// Removes item at the back of the list and returns nothing
METHOD Remove_Last : I_Write_Only_List
VAR_OUTPUT
	bSuccess : BOOL;
END_VAR
END_METHOD

// Manually resize list. If list becomes smaller, item on higher locations will be deleted.
METHOD Resize : I_Write_Only_List
VAR_INPUT
	nSize : DINT; // New size of list.
END_VAR
VAR_OUTPUT
	bSuccess : BOOL;
END_VAR
END_METHOD

// Reverses the order of items in the list
METHOD Reverse : I_Write_Only_List
VAR_OUTPUT
	bSuccess : BOOL;
END_VAR
END_METHOD

// Adds new item to list in the specified location without resizing list
METHOD Set : I_Write_Only_List
VAR_INPUT
	Item 	: ANY; 	// Item to store in list
	nIndex 	: DINT; // Location of item
END_VAR
VAR_OUTPUT
	bSuccess : BOOL;
END_VAR
END_METHOD

END_INTERFACE

// POUs/Examples/P_Example_Array_List
PROGRAM INTERNAL P_Example_Array_List
VAR
	eState 		: (IDLE, INSERT, REVERSE, RESIZE, GET, SET, FIND, CLEAR, ADD_FRONT, ADD_BACK, REMOVE, REMOVE_AT);
	fbArray_List: FB_Array_List(2);
	nFind 		: T_Capacity;
	sData 		: WSTRING;
	sRTNData	: ARRAY[0..6] OF WSTRING;
	nCount 		: T_Capacity;
	stError 	: ST_ERROR;
	bSuccess 	: BOOL;
END_VAR

stError := fbArray_List._Error_Status;
CASE eState OF
	INSERT:
		sData := "Cats";	fbArray_List.Insert(sData, 0);
		sData := "Dogs";	fbArray_List.Insert(sData, 1);
		sData := "Ravens";	fbArray_List.Insert(sData, 2);
		sData := "Mollies";	fbArray_List.Insert(sData, 3);
	REVERSE:
		fbArray_List.Reverse();
	RESIZE:
		fbArray_List.Resize(3);
	GET: 
		Scrub();
		fbArray_List
			.Get(sRTNData[0], 0)
			.Get(sRTNData[1], 1)
			.Get(sRTNData[2], 2)
			.Get(sRTNData[3], 3)
			.Get(sRTNData[4], 4)
			.Get(sRTNData[5], 5)
			.Get(sRTNData[6], 6);
	SET:
		sData := "Ravens";	fbArray_List.Set(sData, 0);
		sData := "Mollies";	fbArray_List.Set(sData, 1);
		sData := "Dogs";	fbArray_List.Set(sData, 2);
		sData := "Cats";	fbArray_List.Set(sData, 3);
	FIND:
		sData := "Dogs"; fbArray_List.Find(sData, nIndex => nFind);
	CLEAR:
		fbArray_List.Clear();
	ADD_FRONT:
		sData := "Pythons";fbArray_List.Add_Front(sData);
	ADD_BACK:
		sData := "Anacondas"; fbArray_List.Add_Back(sData);
	REMOVE:
		fbArray_List.Remove(bSuccess => bSuccess);
	REMOVE_AT:
		fbArray_List.Remove_At(2);
		
END_CASE
nCount := fbArray_List._Count;
eState := IDLE;

METHOD PRIVATE Scrub
VAR
	i 			: T_Capacity;
END_VAR
FOR i := 0 TO SIZEOF(sRTNData)/SIZEOF(sRTNData[0])-1 DO sRTNData[i] := ""; END_FOR
END_METHOD

END_PROGRAM

// POUs/Function Blocks/FB_Array_List
(* A dynamic array that holds data of multiple types and can grow or shrink at run time. *)
{attribute 'enable_dynamic_creation'}
{attribute 'no_assign'}
FUNCTION_BLOCK FB_Array_List EXTENDS FB_Collection IMPLEMENTS I_List, I_Generic_List
VAR
	pData 		: POINTER TO ST_GENERIC;
END_VAR
VAR CONSTANT
	//{warning disable C0228}
	stData 		: ST_GENERIC := (TypeClass := __SYSTEM.TYPE_CLASS.TYPE_NONE);
END_VAR

// Raises an expection if list is empty
METHOD PROTECTED EmptyListException : BOOL
VAR_INPUT
END_VAR
IF THIS^._Is_Empty THEN
	stError.bSTATUS := TRUE;
	stError.nCODE 	:= 2936;
	stError.sSOURCE := 'List is empty';
ELSE
	This^.ClearException();
	END_IF
EmptyListException := stError.bSTATUS;
END_METHOD

METHOD PROTECTED LessThanZeroException : BOOL
VAR_INPUT
	nIndex : DINT;
END_VAR
IF (nIndex < 0) THEN
	stError.bSTATUS := TRUE;
	stError.nCODE 	:= 5365;
	stError.sSOURCE := 'Out of bounds. Index is less than zero.';
ELSE
	This^.ClearException();
	END_IF
LessThanZeroException := stError.bSTATUS;
END_METHOD

// Compares memory sizes of 2 addresses. Returns TRUE  and raises error flag if theyre not same size.
METHOD PROTECTED MemCmpErrExpection : BOOL
VAR_INPUT
	pDestAddr,
	pSrcAddr 	: PVOID;
	nSize 		: UDINT;
END_VAR
VAR_INST
	nMemErr : DINT;
END_VAR
nMemErr := MEMCMP(pDestAddr, pSrcAddr, nSize);
IF nMemErr = -1 THEN 
	stError.bSTATUS := TRUE;
	stError.nCODE 	:= 4129;
	stError.sSOURCE := 'Incorrect parameter values. Destination address smaller than source address';
	
ELSIF nMemErr = 0 THEN THIS^.ClearException();
	
ELSIF nMemErr = 1 THEN
	stError.bSTATUS := TRUE;
	stError.nCODE 	:= 4823;
	stError.sSOURCE := 'Incorrect parameter values. Destination address greater that source address';

ELSE
	stError.bSTATUS := TRUE;
	stError.nCODE 	:= 4564;
	stError.sSOURCE := 'Incorrect parameter values. Pointer to destination/source address is NULL or allocated address memory is NULL.';
	END_IF

MemCmpErrExpection := stError.bSTATUS;
END_METHOD

METHOD PROTECTED OutOfBoundsException : BOOL
VAR_INPUT
	nIndex : DINT;
END_VAR
IF (nIndex < 0) OR (nIndex >= THIS^._Count) THEN
	stError.bSTATUS := TRUE;
	stError.nCODE 	:= 5374;
	stError.sSOURCE := 'Out of bounds. You tried to access data outside the range of this list.';
ELSE
	This^.ClearException();
	END_IF
OutOfBoundsException := stError.bSTATUS;
END_METHOD

METHOD TypeMismatchException : BOOL
VAR_INPUT
	Dest,
	Src 	: __SYSTEM.AnyType;
END_VAR
IF Dest.diSize <> Src.diSize THEN
	stError.bSTATUS := TRUE;
	stError.nCODE 	:= 3172;
	stError.sSOURCE := 'Type mismatch. Byte sizes are not the same';
ELSIF Dest.TypeClass <> Src.TypeClass THEN
	stError.bSTATUS := TRUE;
	stError.nCODE 	:= 3172;
	stError.sSOURCE := 'Type mismatch. Type classes are not the same';
ELSE
	THIS^.ClearException();
END_IF
TypeMismatchException := stError.bSTATUS;
END_METHOD

// Copy data from source memory space to desination memory space
METHOD PROTECTED CopyValueTo
VAR_INPUT
	Dest, Src 	: T_Generic;
END_VAR
MEMMOVE(Dest.pValue, Src.pValue, TO_UDINT(Src.diSize));
END_METHOD

// Decrement list size by 1.
METHOD PROTECTED DecrementCount
THIS^.nCount := THIS^.nCount - 1;
END_METHOD

// Deletes/frees Generic value's value from memory
METHOD PROTECTED Free_Value
VAR_INPUT
	Variable : T_Generic;
END_VAR
IF Variable.pValue = 0 THEN RETURN; END_IF
__DELETE(Variable.pValue);
END_METHOD

METHOD PROTECTED GetValueAsString : T_MaxString
VAR_INPUT
	 Value : T_Generic;
END_VAR
VAR	
	pBool			: POINTER TO BOOL;
    pByte			: POINTER TO BYTE;
    pWord			: POINTER TO WORD;
    pDWord			: POINTER TO DWORD;
    pLWord			: POINTER TO LWORD;
    pSint			: POINTER TO SINT;
    pInt			: POINTER TO INT;
    pDint			: POINTER TO DINT;
    pLint			: POINTER TO LINT;
    pUSint			: POINTER TO USINT;
    pUInt			: POINTER TO UINT;
    pUDint			: POINTER TO UDINT;
    pULint			: POINTER TO ULINT;
    pReal			: POINTER TO REAL;
    pLReal			: POINTER TO LREAL;
    pString			: POINTER TO STRING(255);
    pWString		: POINTER TO WSTRING;
    pTime			: POINTER TO TIME;
    pDate			: POINTER TO DATE;
    pDate_And_Time	: POINTER TO DATE_AND_TIME;
    pTime_Of_Day	: POINTER TO TIME_OF_DAY;
    pPointer		: PVOID;
	pLTime 			: POINTER TO LTIME;
END_VAR
IF Value.pValue = 0 THEN GetValueAsString := 'NULL'; RETURN; END_IF;

CASE Value.TypeClass OF 
	__SYSTEM.TYPE_CLASS.TYPE_BOOL:
		pBool := Value.pValue;
		GetValueAsString := TO_STRING(pBool^);
		
    __SYSTEM.TYPE_CLASS.TYPE_BYTE:
		pByte := Value.pValue;
		GetValueAsString := TO_STRING(pByte^);
		
    __SYSTEM.TYPE_CLASS.TYPE_WORD:
		pWord := Value.pValue;
		GetValueAsString := TO_STRING(pWord^);
		
    __SYSTEM.TYPE_CLASS.TYPE_DWORD:
		pDWord := Value.pValue;
		GetValueAsString := TO_STRING(pDWord^);
		
    __SYSTEM.TYPE_CLASS.TYPE_LWORD:
		pLWord := Value.pValue;
		GetValueAsString := TO_STRING(pLWord^);
		
    __SYSTEM.TYPE_CLASS.TYPE_SINT:
		pSint := Value.pValue;
		GetValueAsString := TO_STRING(pSint^);
		
    __SYSTEM.TYPE_CLASS.TYPE_INT:
		pInt := Value.pValue;
		GetValueAsString := TO_STRING(pInt^);
		
    __SYSTEM.TYPE_CLASS.TYPE_DINT:
		pDint := Value.pValue;
		GetValueAsString := TO_STRING(pDint^);
		
    __SYSTEM.TYPE_CLASS.TYPE_LINT:
		pLint := Value.pValue;
		GetValueAsString := TO_STRING(pLint^);
		
    __SYSTEM.TYPE_CLASS.TYPE_USINT:
		pUSint := Value.pValue;
		GetValueAsString := TO_STRING(pUSint^);
		
    __SYSTEM.TYPE_CLASS.TYPE_UINT:
		pUInt := Value.pValue;
		GetValueAsString := TO_STRING(pUInt^);
		
    __SYSTEM.TYPE_CLASS.TYPE_UDINT:
		pUDint := Value.pValue;
		GetValueAsString := TO_STRING(pUDint^);
		
    __SYSTEM.TYPE_CLASS.TYPE_ULINT:
		pULint := Value.pValue;
		GetValueAsString := TO_STRING(pULint^);
		
   __SYSTEM.TYPE_CLASS.TYPE_REAL:
		pReal := Value.pValue;
		GetValueAsString := TO_STRING(pReal^);
		
    __SYSTEM.TYPE_CLASS.TYPE_LREAL:
		pLReal := Value.pValue;
		GetValueAsString := TO_STRING(pLReal^);
		
    __SYSTEM.TYPE_CLASS.TYPE_STRING:
		pString := Value.pValue;
		GetValueAsString := TO_STRING(pString^);
		
   __SYSTEM.TYPE_CLASS.TYPE_WSTRING:
		pWString := Value.pValue;
		GetValueAsString := TO_STRING(pWString^);
		
    __SYSTEM.TYPE_CLASS.TYPE_TIME:
		pTime := Value.pValue;
		GetValueAsString := TO_STRING(pTime^);
		
    __SYSTEM.TYPE_CLASS.TYPE_DATE:
		pDate := Value.pValue;
		GetValueAsString := TO_STRING(pDate^);
		
    __SYSTEM.TYPE_CLASS.TYPE_DATEANDTIME:
		pDate_And_Time := Value.pValue;
		GetValueAsString := TO_STRING(pDate_And_Time^);
		
    __SYSTEM.TYPE_CLASS.TYPE_TIMEOFDAY:
		pTime_Of_Day := Value.pValue;
		GetValueAsString := TO_STRING(pTime_Of_Day^);
	
	__SYSTEM.TYPE_CLASS.TYPE_POINTER:
		GetValueAsString := TO_STRING(Value.pValue);
		
	__SYSTEM.TYPE_CLASS.TYPE_LTIME:
		pLTime := Value.pValue;
		GetValueAsString := TO_STRING(pLTime^);
ELSE
	GetValueAsString := 'TYPE TO STRING CONVERSION NOT SUPPORTED BY THIS TYPE'; 
END_CASE
END_METHOD

// Increments list size by 1
METHOD PROTECTED IncrementCount
VAR_INPUT
END_VAR
THIS^.nCount := THIS^.nCount + 1;
END_METHOD

// Adds an item to the end of the list
METHOD PROTECTED Internal_Add_Back
VAR_INPUT
	Item 		: T_Generic; // Item to store in list
END_VAR
VAR_OUTPUT
	bSuccess 	: BOOL;
END_VAR
IF THIS^._Is_Empty THEN THIS^.FB_init(FALSE,FALSE, 1); THIS^.Internal_Set(Item, 0, bSuccess => bSuccess); RETURN; END_IF
THIS^.Resize(THIS^._Count+1);
THIS^.Free_Value(THIS^.pData[THIS^._Count-1]);
THIS^.pData[THIS^._Count-1] := THIS^.Malloc_Value(Item);
THIS^.CopyValueTo(THIS^.pData[THIS^._Count-1], Item);
bSuccess := TRUE;
END_METHOD

// Adds an item at the front of the list
METHOD PROTECTED Internal_Add_Front
VAR_INPUT
	Item 	 : ANY; // Item to store in list
END_VAR
VAR_OUTPUT
	bSuccess : BOOL;
END_VAR
VAR
	pOld_Data : POINTER TO ST_GENERIC;
	i : DINT;
END_VAR
IF THIS^._Is_Empty THEN THIS^.FB_init(FALSE,FALSE, 1); THIS^.Internal_Set(Item, 0, bSuccess => bSuccess); RETURN; END_IF

pOld_Data := THIS^.pData;
THIS^.pData := THIS^.Malloc_Array(THIS^._Count+1);

FOR i := 1 TO THIS^._Count DO
	THIS^.pData[i] := THIS^.Malloc_Value(pOld_Data[i-1]);
	THIS^.CopyValueTo(THIS^.pData[i], pOld_Data[i-1]);
	THIS^.Free_Value(pOld_Data[i-1]);
	END_FOR
__DELETE(pOld_Data);
THIS^.Internal_Set(Item, 0);
THIS^.IncrementCount();
bSuccess := TRUE;
END_METHOD

// Adds new item to list in the specified location without resizing list
METHOD PROTECTED Internal_Set
VAR_INPUT
	Item 	: T_Generic; 	// Item to store in list
	nIndex 	: T_Capacity; // Location of item
END_VAR
VAR_OUTPUT
	bSuccess : BOOL;
END_VAR
IF THIS^.OutOfBoundsException(nIndex) OR THIS^.EmptyListException() THEN RETURN; END_IF
THIS^.Free_Value(THIS^.pData[nIndex]);
THIS^.pData[nIndex] := THIS^.Malloc_Value(Item);
THIS^.CopyValueTo(THIS^.pData[nIndex], Item);
bSuccess := TRUE;
END_METHOD

// Allocate memory space for Array of Generics on the heap, returns Pointer to start of Generic Array;
// WARNING!!! Always have a place to store the return otherwise a memory leak will occur.
METHOD PROTECTED Malloc_Array : POINTER TO ST_GENERIC
VAR_INPUT
	nSize : T_Capacity; // Array Size
END_VAR
VAR
	i, nByte_Size: T_Capacity;
END_VAR
VAR CONSTANT
	stData 		: T_Generic_Ex := ();
END_VAR
nByte_Size := SIZEOF(T_Generic_Ex)*nSize;
Malloc_Array := __NEW(BYTE, TO_UDINT(nByte_Size));
END_METHOD

// Allocate memory space for the Generic value's data on the heap, returns Generic;
// WARNING!!! Always have a place to store the return otherwise a memory leak will occur.
METHOD PROTECTED Malloc_Value : ST_GENERIC
VAR_INPUT
	Variable : T_Generic;
END_VAR
Malloc_Value.sValue 	:= THIS^.GetValueAsString(Variable);
Malloc_Value.pValue 	:= __NEW(BYTE, TO_UDINT(Variable.diSize)); // Allocate space in memory to store data value.
Malloc_Value.diSize 	:= Variable.diSize;
Malloc_Value.TypeClass 	:= Variable.TypeClass;
END_METHOD

(* Set value of __SYSTEM.Anytype variable *)
METHOD PROTECTED SetValue
VAR_INPUT
	Variable	: T_Generic;
	Value 		: USINT; // Character/byte to set.
END_VAR
MEMSET(Variable.pValue, Value, TO_UDINT(Variable.diSize));
END_METHOD

(* Checks of list is empty.*)
PROPERTY _Is_Empty : BOOL
GET
_Is_Empty := THIS^.nCount = 0;
END_GET
END_PROPERTY

// Adds an item to the end of the list
METHOD Add_Back : I_List
VAR_INPUT
	Item 	: ANY; // Item to store in list
END_VAR
VAR_OUTPUT
	bSuccess : BOOL;
END_VAR
Add_Back := THIS^;
IF THIS^._Is_Empty THEN THIS^.FB_init(FALSE,FALSE, 1); THIS^.Set(Item, 0, bSuccess => bSuccess); RETURN; END_IF
THIS^.Resize(THIS^._Count+1);
THIS^.Free_Value(THIS^.pData[THIS^._Count-1]);
THIS^.pData[THIS^._Count-1] := THIS^.Malloc_Value(Item);
THIS^.CopyValueTo(THIS^.pData[THIS^._Count-1], Item);
bSuccess := TRUE;
END_METHOD

// Adds an item at the front of the list
METHOD Add_Front : I_List
VAR_INPUT
	Item 	 : ANY; // Item to store in list
END_VAR
VAR_OUTPUT
	bSuccess : BOOL;
END_VAR
VAR
	pOld_Data : POINTER TO ST_GENERIC;
	i : DINT;
END_VAR
Add_Front := THIS^;
IF THIS^._Is_Empty THEN THIS^.FB_init(FALSE,FALSE, 1); THIS^.Set(Item, 0, bSuccess => bSuccess); RETURN; END_IF

pOld_Data := THIS^.pData;
THIS^.pData := THIS^.Malloc_Array(THIS^._Count+1);

FOR i := 1 TO THIS^._Count DO
	THIS^.pData[i] := THIS^.Malloc_Value(pOld_Data[i-1]);
	THIS^.CopyValueTo(THIS^.pData[i], pOld_Data[i-1]);
	THIS^.Free_Value(pOld_Data[i-1]);
	END_FOR
__DELETE(pOld_Data);
THIS^.Set(Item, 0);
THIS^.IncrementCount();
bSuccess := TRUE;
END_METHOD

// Empties/Clears/Deletes every item in the list
METHOD Clear
VAR
	i : DINT;
END_VAR
IF NOT(THIS^._Is_Empty) THEN 
	FOR i := 0 TO THIS^._Count - 1 DO THIS^.Free_Value(THIS^.pData[i]); END_FOR
	__DELETE(THIS^.pData); 
	THIS^.nCount := 0; 
	END_IF
END_METHOD

(* Checks if item is contained in list *)
METHOD Contains : BOOL
VAR_INPUT
	Item : ANY; // Item to find in list
END_VAR
THIS^.Find(Item, bSuccess => Contains);
END_METHOD

METHOD FB_exit : BOOL
VAR_INPUT
	bInCopyCode : BOOL; // if TRUE, the exit method is called for exiting an instance that is copied afterwards (online change).
END_VAR
THIS^.Clear();
END_METHOD

METHOD FB_init : BOOL
VAR_INPUT
	bInitRetains 	: BOOL; 		// if TRUE, the retain variables are initialized (warm start / cold start)
	bInCopyCode 	: BOOL; 		// if TRUE, the instance afterwards gets moved into the copy code (online change)
	nLength 		: T_Capacity;	// Length to initialise array with.
END_VAR
VAR
	i, nByte_Size 	: DINT;
END_VAR
THIS^.Clear();
IF nLength <= 0 THEN RETURN; END_IF
THIS^.nCount := nLength;
THIS^.pData := THIS^.Malloc_Array(nLength);
END_METHOD

// Find the location of an item in list.
METHOD Find : I_List
VAR_INPUT
	Item 		: ANY; // Item to find in list
END_VAR
VAR_OUTPUT
	nIndex		: T_Capacity; //Location of item in list 
	bSuccess 	: BOOL;
END_VAR
VAR
	i : DINT;
	n : DINT := -1;
END_VAR
Find := THIS^;
IF THIS^.EmptyListException() THEN nIndex := -1; RETURN; END_IF
FOR i := 0 TO THIS^._Count-1 DO
	IF (THIS^.pData[i].pValue = 0) 					 THEN CONTINUE; END_IF
	IF (Item.TypeClass <> THIS^.pData[i].TypeClass) THEN CONTINUE; END_IF
	IF (Item.pValue^ <> THIS^.pData[i].pValue^) 	 THEN CONTINUE; END_IF
	
	CASE Item.TypeClass OF
		__SYSTEM.TYPE_CLASS.TYPE_STRING:
			IF LEN2(Item.pValue) <> LEN2(THIS^.pData[i].pValue) THEN CONTINUE; END_IF
			n := MEMCMP(Item.pValue, THIS^.pData[i].pValue, LEN2(THIS^.pData[i].pValue)+1);
				
		__SYSTEM.TYPE_CLASS.TYPE_WSTRING:
			IF WLEN2(Item.pValue) <> WLEN2(THIS^.pData[i].pValue) THEN CONTINUE; END_IF
			n := MEMCMP(Item.pValue, THIS^.pData[i].pValue, (WLEN2(THIS^.pData[i].pValue)*SIZEOF(WORD))+1);
	ELSE
		IF (Item.diSize <> THIS^.pData[i].diSize) THEN CONTINUE; END_IF	
		n := MEMCMP(Item.pValue, THIS^.pData[i].pValue, TO_UDINT(Item.diSize));
		END_CASE
		IF n = 0 THEN nIndex := i; bSuccess := TRUE; RETURN; END_IF
	END_FOR
nIndex := -1;
END_METHOD

// Gets item at specified location;
METHOD Get : I_List
VAR_INPUT
	Return_Item 	: ANY;  // Variable to store requested node value
	nIndex 			: T_Capacity; // Location of node
END_VAR
VAR_OUTPUT
	bSuccess 		: BOOL;
END_VAR
Get := THIS^;
IF THIS^.EmptyListException() OR THIS^.OutOfBoundsException(nIndex) THEN RETURN; END_IF
IF THIS^.TypeMismatchException(Return_Item, THIS^.pData[nIndex]) THEN RETURN; END_IF
THIS^.CopyValueTo(Return_Item, THIS^.pData[nIndex]);
bSuccess := TRUE;
END_METHOD

// Gets item at the front of the list 
METHOD Get_First : I_List
VAR_INPUT
	Return_Item 	: ANY; // Variable to store returned item
END_VAR
VAR_OUTPUT
	bSuccess : BOOL;
END_VAR
Get_First := THIS^;
THIS^.Get(Return_Item, 0, bSuccess => bSuccess);
END_METHOD

// Gets a value from a list in it's generic form.
// (* Use carefully as this contains the pointer of the actual value in the collection. *)
// If you wish to use this it is recommeded you create a copy of the returned value using MEMMOVE or MEMCPY
METHOD Get_Generic : I_Generic_List
VAR_INPUT
	nIndex 		: T_Capacity; 	// Location of item
END_VAR
VAR_OUTPUT
	Return_Item : T_Generic;  	// Variable to store returned item
	bSuccess 	: BOOL;
END_VAR
Get_Generic := THIS^;
IF THIS^.EmptyListException() OR THIS^.OutOfBoundsException(nIndex) THEN RETURN; END_IF
Return_Item := THIS^.pData[nIndex];
bSuccess := TRUE;
END_METHOD

// Gets item at the back of the list 
METHOD Get_Last : I_List
VAR_INPUT
	Return_Item 	: ANY; // Variable to store returned item
END_VAR
VAR_OUTPUT
	bSuccess : BOOL;
END_VAR
Get_Last := THIS^;
THIS^.Get(Return_Item, THIS^._Count - 1, bSuccess => bSuccess);
END_METHOD

// Returns item as a string, if type to string conversion is supported
METHOD Get_Value_As_String : I_List
VAR_INPUT
	nIndex	: T_Capacity; // Location of item
END_VAR
VAR_OUTPUT
	sItem 	: T_MaxString; // Variable to store returned item
END_VAR
Get_Value_As_String := THIS^;
IF THIS^.EmptyListException() OR THIS^.OutOfBoundsException(nIndex) THEN sItem := 'ERR: List is Empty or index Out of Bounds'; RETURN; END_IF
sItem := THIS^.pData[nIndex].sValue;
END_METHOD

// Adds new item to list at specified location, if index = 0, item will be added at the front, if index = count, item will be added at the back
METHOD Insert : I_List
VAR_INPUT
	Item 	: ANY;  		// Item to store in list
	nIndex 	: T_Capacity; // Location of item
END_VAR
VAR_OUTPUT
	bSuccess : BOOL;
END_VAR
VAR
	pOld_Data 	: POINTER TO T_Generic;
	i 			: T_Capacity;
END_VAR
Insert := THIS^;
IF nIndex = 0 THEN THIS^.Add_Front(Item, bSuccess => bSuccess); RETURN; END_IF
IF nIndex = THIS^._Count THEN THIS^.Add_Back(Item, bSuccess => bSuccess); RETURN; END_IF
IF THIS^.OutOfBoundsException(nIndex) THEN RETURN; END_IF

pOld_Data := THIS^.pData;
THIS^.pData := THIS^.Malloc_Array(THIS^._Count+1);
THIS^.IncrementCount();

FOR i := 0 TO nIndex-1 DO
	THIS^.pData[i] := THIS^.Malloc_Value(pOld_Data[i]);
	THIS^.CopyValueTo(THIS^.pData[i], pOld_Data[i]);
	THIS^.Free_Value(pOld_Data[i]);
	END_FOR
	
THIS^.Set(Item, nIndex, bSuccess => bSuccess);
	
FOR i := nIndex+1 TO THIS^._Count-1 DO
	THIS^.pData[i] := THIS^.Malloc_Value(pOld_Data[i-1]);
	THIS^.CopyValueTo(THIS^.pData[i], pOld_Data[i-1]);
	THIS^.Free_Value(pOld_Data[i-1]);
	END_FOR
__DELETE(pOld_Data);
END_METHOD

// Adds new item to list at specified location using the generic form. 
// If index = 0, item will be added at the front, if index = count, item will be added at the back
METHOD Insert_Generic : I_Generic_List
VAR_INPUT
	Item 	: T_Generic;  	// Item to store in list
	nIndex 	: T_Capacity; 			// Location of item
END_VAR
VAR_OUTPUT
	bSuccess : BOOL;
END_VAR
VAR
	pOld_Data 	: POINTER TO T_Generic;
	i 			: T_Capacity;
END_VAR
Insert_Generic := THIS^;

// Add to front
IF nIndex = 0 THEN THIS^.Internal_Add_Front(Item, bSuccess => bSuccess); RETURN; END_IF

// Add to back
IF nIndex = THIS^._Count THEN Internal_Add_Back(Item, bSuccess => bSuccess); RETURN; END_IF

IF THIS^.OutOfBoundsException(nIndex) THEN RETURN; END_IF

pOld_Data := THIS^.pData;
THIS^.pData := THIS^.Malloc_Array(THIS^._Count+1);
THIS^.IncrementCount();

FOR i := 0 TO nIndex-1 DO
	THIS^.pData[i] := THIS^.Malloc_Value(pOld_Data[i]);
	THIS^.CopyValueTo(THIS^.pData[i], pOld_Data[i]);
	THIS^.Free_Value(pOld_Data[i]);
	END_FOR

// Set value
Internal_Set(Item, nIndex, bSuccess => bSuccess);
	
FOR i := nIndex+1 TO THIS^._Count-1 DO
	THIS^.pData[i] := THIS^.Malloc_Value(pOld_Data[i-1]);
	THIS^.CopyValueTo(THIS^.pData[i], pOld_Data[i-1]);
	THIS^.Free_Value(pOld_Data[i-1]);
	END_FOR
__DELETE(pOld_Data);
END_METHOD

// Removes item at the front of the list and returns nothing
METHOD Remove : I_List
VAR_OUTPUT
	bSuccess : BOOL;
END_VAR
VAR
	i : DINT;
	pOld_Data 	: POINTER TO ST_GENERIC;
END_VAR
//// New ///
Remove := THIS^;
IF THIS^.EmptyListException() THEN RETURN; END_IF
IF THIS^._Count = 1 THEN THIS^.Clear(); bSuccess := TRUE; RETURN; END_IF;

THIS^.Free_Value(THIS^.pData[0]);
pOld_Data := pData;
pData := THIS^.Malloc_Array(THIS^._Count - 1);
FOR i := 1 TO THIS^._Count - 1 DO
	pData[i-1] := pOld_Data[i];
	END_FOR

__DELETE(pOld_Data);
THIS^.DecrementCount();
bSuccess := TRUE;
END_METHOD

// Remove item at specified location and return nothing
METHOD Remove_At : I_List
VAR_INPUT
	nIndex : T_Capacity; // Location of item
END_VAR
VAR_OUTPUT
	bSuccess : BOOL;
END_VAR
VAR
	i : DINT;
END_VAR
Remove_At := THIS^;
IF THIS^.EmptyListException() THEN RETURN; END_IF
IF THIS^.OutOfBoundsException(nIndex) THEN RETURN; END_IF
IF nIndex = 0 THEN THIS^.Remove(bSuccess => bSuccess); RETURN; END_IF
IF nIndex = THIS^._Count - 1 THEN THIS^.Resize(THIS^._Count - 1, bSuccess => bSuccess); RETURN; END_IF
THIS^.Free_Value(THIS^.pData[nIndex]);
FOR i := nIndex TO THIS^._Count-1 DO THIS^.pData[i] := THIS^.pData[i+1]; END_FOR
THIS^.Resize(THIS^._Count-1, bSuccess => bSuccess);
END_METHOD

// Removes item at the back of the list and returns nothing
METHOD Remove_Last : I_List
VAR_OUTPUT
	bSuccess : BOOL;
END_VAR
Remove_Last := THIS^;
THIS^.Remove_At(THIS^._Count-1, bSuccess => bSuccess);
END_METHOD

// Manually resize list. If list becomes smaller, items on higher locations will be deleted.
METHOD Resize : I_List
VAR_INPUT
	nSize : T_Capacity; // New size of list.
END_VAR
VAR_OUTPUT
	bSuccess : BOOL;
END_VAR
VAR
	pOld_Data 		: POINTER TO ST_GENERIC;
	i,
	nOld_Data_Count, 
	nByte_Size : DINT;
END_VAR
Resize := THIS^;
IF THIS^.LessThanZeroException(nSize) THEN RETURN; END_IF
IF (nSize = 0) THEN THIS^.Clear(); RETURN; END_IF
IF nSize = THIS^._Count THEN RETURN; END_IF

bSuccess := TRUE;

IF THIS^._Is_Empty THEN THIS^.FB_init(FALSE,FALSE, nSize); RETURN; END_IF

pOld_Data 		:= THIS^.pData;
nOld_Data_Count := THIS^._Count;

THIS^.pData := THIS^.Malloc_Array(nSize);

FOR i := 0 TO nSize - 1 DO
	IF (i = nOld_Data_Count) AND (nSize > nOld_Data_Count) THEN EXIT; END_IF
	THIS^.pData[i] := THIS^.Malloc_Value(pOld_Data[i]);
	THIS^.CopyValueTo(THIS^.pData[i], pOld_Data[i]);
	THIS^.Free_Value(pOld_Data[i]);
	END_FOR
__DELETE(pOld_Data);
THIS^.nCount := nSize;

bSuccess := TRUE;
END_METHOD

// Reverses the order of items in the list
METHOD Reverse : I_List
VAR_OUTPUT
	bSuccess : BOOL;
END_VAR
VAR
	pOld_Data 	: POINTER TO ST_GENERIC;
	nByte_Size 	: DINT;
	i			: DINT;
END_VAR
Reverse := THIS^;
IF THIS^.EmptyListException() THEN RETURN; END_IF
IF THIS^._Count = 1 THEN RETURN; END_IF

pOld_Data 	:= THIS^.pData;

THIS^.pData := THIS^.Malloc_Array(THIS^._Count);

FOR i:= 0 TO THIS^._Count - 1 DO
	THIS^.pData[i] := THIS^.Malloc_Value(pOld_Data[(THIS^._Count-1)-i]);
	THIS^.CopyValueTo(THIS^.pData[i], pOld_Data[(THIS^._Count-1)-i]);
	THIS^.Free_Value(pOld_Data[(THIS^._Count-1)-i]);
	END_FOR
__DELETE(pOld_Data);

bSuccess := TRUE;
END_METHOD

// Adds new item to list in the specified location without resizing list
METHOD Set : I_List
VAR_INPUT
	Item 	: ANY; 	// Item to store in list
	nIndex 	: T_Capacity; // Location of item
END_VAR
VAR_OUTPUT
	bSuccess : BOOL;
END_VAR
Set := THIS^;
IF THIS^.OutOfBoundsException(nIndex) OR THIS^.EmptyListException() THEN RETURN; END_IF
THIS^.Free_Value(THIS^.pData[nIndex]);
THIS^.pData[nIndex] := THIS^.Malloc_Value(Item);
THIS^.CopyValueTo(THIS^.pData[nIndex], Item);
bSuccess := TRUE;
END_METHOD

END_FUNCTION_BLOCK

// POUs/Function Blocks/FB_Collection
FUNCTION_BLOCK ABSTRACT FB_Collection IMPLEMENTS I_Collection
VAR
	nCount 	: T_Capacity; // Size of Collection
	stError : T_Error := F_Error(FALSE, GVL_CmpErrors.ERR_OK,'');
END_VAR

METHOD PROTECTED ClearException : BOOL
VAR_INPUT
END_VAR
THIS^.stError := F_Error(FALSE, 0, '');
END_METHOD

// Raises an expection if list is empty
METHOD PROTECTED EmptyListException : BOOL
VAR_INPUT
END_VAR
IF THIS^._Is_Empty THEN THIS^.RaiseException(2936, 'Collection is empty'); EmptyListException := TRUE; END_IF
END_METHOD

METHOD PROTECTED FailedInsertionException : BOOL
VAR_INPUT
END_VAR
THIS^.RaiseException(2667, 'Failed to insert item into collection');
END_METHOD

METHOD PROTECTED NullReferenceException : BOOL
THIS^.RaiseException(2000+GVL_CmpErrors.ERR_INVALID_REFERENCE, 'Null or Invalid Reference');
END_METHOD

METHOD PROTECTED OutOfBoundsException : BOOL
VAR_INPUT
	nIndex : T_Capacity;
END_VAR
IF (nIndex < 0) OR (nIndex >= THIS^._Count) THEN
	THIS^.RaiseException(2374,'Out of bounds. You tried to access data outside the range of this collection.');
	OutOfBoundsException := TRUE;
	END_IF
END_METHOD

METHOD PROTECTED RaiseException : BOOL
VAR_INPUT
	nCode 	: DINT;
	sSource : T_MaxString;
END_VAR
THIS^.stError := F_Error(TRUE, nCode, sSource);
END_METHOD

METHOD PROTECTED ValueFoundException : BOOL
VAR_INPUT
END_VAR
THIS^.RaiseException(2748, 'Value is contained in collection');
END_METHOD

METHOD PROTECTED ValueNotFoundException : BOOL
VAR_INPUT
END_VAR
THIS^.RaiseException(2923, 'Value is not contain in collection');
END_METHOD

// Clears value by setting it's entire memory space to NULL
METHOD PROTECTED ClearValue
VAR_INPUT
	Value : __SYSTEM.AnyType;
END_VAR
MEMSET(Value.pValue, 16#0, TO_UDINT(Value.diSize));
END_METHOD

// Copy data from source memory space to desination memory space
METHOD PROTECTED CopyValueTo
VAR_INPUT
	Dest, Src : __SYSTEM.AnyType;
END_VAR
THIS^.ClearValue(Dest);
MEMMOVE(Dest.pValue, Src.pValue, TO_UDINT(MIN(Dest.diSize, Src.diSize)));
END_METHOD

// Decrement list size by 1.
METHOD PROTECTED DecrementCount
VAR_INPUT
END_VAR
THIS^.nCount := THIS^.nCount - 1;
END_METHOD

// Increments list size by 1
METHOD PROTECTED IncrementCount
VAR_INPUT
END_VAR
THIS^.nCount := THIS^.nCount + 1;
END_METHOD

(* Number of elements in collection*)
PROPERTY _Count : T_Capacity
GET
_Count := THIS^.nCount;
END_GET
END_PROPERTY

(* Gets collection's error status *)
PROPERTY _Error_Status : T_Error
GET
_Error_Status := THIS^.stError;
END_GET
SET
PROTECTED 
VAR
END_VAR
THIS^.stError := THIS^.stError;
END_SET
END_PROPERTY

(* Checks if collection is empty.*)
PROPERTY _Is_Empty : BOOL
GET
_Is_Empty := THIS^._Count = 0;
END_GET
END_PROPERTY

(* Empties/Clears/Deletes every element on the collection*)
METHOD Clear
END_METHOD

END_FUNCTION_BLOCK

// POUs/Functions/F_Error
// Error Function: Passes error code and message to type ST_ERROR when bStatus = TRUE.  
FUNCTION F_Error : T_Error
VAR_INPUT
	bStatus : BOOL; 		// Trigger to pass code and message | Note: Default is FALSE
	nCode 	: DINT; 		// Code to pass to error struct | Note: code is 0 if there is no error
	sSource : T_MaxString; 	// Message to pass to error struct | Note: message is 'No Error.'  if there is no error
END_VAR
VAR
END_VAR

F_Error.bSTATUS := bStatus; 
IF bStatus THEN F_Error.nCODE := nCode; F_Error.sSOURCE := sSource;
ELSE F_Error.nCODE := GVL_CmpErrors.ERR_OK; F_Error.sSOURCE := 'No Error'; END_IF

END_FUNCTION

// POUs/Examples/P_Example_Binary_Search_Tree
PROGRAM INTERNAL P_Example_Binary_Search_Tree
VAR
	eState 		: (IDLE, INSERT, FIND, REMOVE, TRAVERSE, CLEAR, CLEAR_LIST, BALANCE);
	fbBST 		: FB_Binary_Search_Tree(T_Type.TYPE_DINT);
	eTrav 		: T_BST_Traversal;
	fbList 		: FB_List;
	arsVal 		: ARRAY[0..20] OF T_MaxString;
	nFind 		: DINT; // Value to find
	bFound 		: BOOL; 
	nRemove 	: DINT; // Value to remove
	bRemoved 	: BOOL;
	arValues	: ARRAY[0..7] OF DINT := [1,2,3,4,5,6,7,8];
	nCount,i 	: DINT;
	stError 	: ST_ERROR;
	sz 			: UDINT;
END_VAR

stError := fbBST._Error_Status;
sz := SIZEOF(fbBST);
nCount := fbBST._Count;
CASE eState OF
	INSERT:
		FOR i := 0 TO (SIZEOF(arValues)/SIZEOF(DINT))-1 DO fbBST.Insert(arValues[i]);END_FOR
				
	FIND:
		fbBST.Find(nFind, bFound => bFound);
		
	REMOVE:
		fbBST.Remove(nRemove, bSuccess => bRemoved);
		
	TRAVERSE:
		fbBST.Traverse(eTrav, fbList);
		FOR i := 0 TO (SIZEOF(arsVal)/SIZEOF(arsVal[0]))-1 DO arsVal[i] := ''; END_FOR
		FOR i := 0 TO fbList._Count-1 DO fbList.Get_Value_As_String(i, sItem => arsVal[i]); END_FOR
					
	CLEAR:
		fbBST.Clear();
		
	CLEAR_LIST:
		fbList.Clear();
		
	BALANCE:
		fbBST.Balance();
END_CASE
eState := IDLE;

END_PROGRAM

// POUs/Function Blocks/FB_Binary_Search_Tree
// Dynamic Binary Search Tree
{attribute 'enable_dynamic_creation'}
{attribute 'no_assign'}
FUNCTION_BLOCK FB_Binary_Search_Tree EXTENDS FB_Collection IMPLEMENTS I_Binary_Search_Tree, I_Generic_Binary_Search_Tree
VAR
	Type_ 		: T_Type;
	pRoot 		: POINTER TO T_BST_Node;
END_VAR

METHOD PROTECTED InvalidTypeException : BOOL
VAR_INPUT
	Data	: T_Generic;
END_VAR
IF THIS^._Type = T_Type.TYPE_ANY THEN RETURN; END_IF
InvalidTypeException := THIS^._Type <> Data.TypeClass;
THIS^.stError := F_Error(InvalidTypeException, GVL_CmpErrors.ERR_TYPE_MISMATCH, 'Invalid input type. Type class not equal to internal type');
END_METHOD

// Checks if bst is ready to be balanced
METHOD PROTECTED Balance_Ready : BOOL
VAR
	nMod 		: T_Capacity;
END_VAR
VAR CONSTANT
	nMod_Const 	: T_Capacity := 4; 
END_VAR
nMod := THIS^._Count MOD nMod_Const;
Balance_Ready := nMod = 0;
END_METHOD

// Compare A to B -> A<B = -1, A=B = 0, A>B = 1
METHOD PROTECTED Compare : DINT
VAR_INPUT
	A, B 	: T_Generic;
END_VAR
VAR
	nSizeA, 
	nSizeB 	: UDINT;
	n 		: DINT; 
END_VAR
CASE A.TypeClass OF
	T_Type.TYPE_STRING:
		nSizeA := LEN2(A.pValue);
		IF (B.TypeClass = T_Type.TYPE_STRING) THEN nSizeB := LEN2(B.pValue)+1; JMP _COMPARE; END_IF
		nSizeB := 0;
			
	T_Type.TYPE_WSTRING:
		nSizeA := WLEN2(A.pValue);
		IF (B.TypeClass = T_Type.TYPE_WSTRING) THEN nSizeB := WLEN2(B.pValue)+1; JMP _COMPARE; END_IF
		nSizeB := 0;
ELSE
	Compare := MEMCMP(A.pValue, B.pValue, TO_UDINT(MIN(A.diSize, B.diSize)));
	RETURN;
END_CASE
_COMPARE:
Compare := MEMCMP(ADR(A), ADR(B), SIZEOF(UDINT));
END_METHOD

METHOD PROTECTED Internal_Find
VAR_INPUT
	Data 		: T_Generic; 	// Generic Data to find
END_VAR
VAR_OUTPUT
	bFound 		: BOOL; // Indicates whether data was found. Found = TRUE, Not Found = FALSE
END_VAR
VAR
	nState 		: DINT;
	pCurrent 	: POINTER TO T_BST_Node;
END_VAR
IF THIS^.pRoot = 0 THEN RETURN; END_IF

pCurrent := THIS^.pRoot;
WHILE pCurrent <> 0 DO
	nState := THIS^.Compare(Data, pCurrent^.Data);
	CASE nState OF
	-1: // Less than
		pCurrent := pCurrent^.pLeft;
	 0: // Equal
	 	bFound := TRUE; EXIT;
	 1: // Greater than
		pCurrent := pCurrent^.pRight;
	ELSE
		EXIT;
	END_CASE
	END_WHILE
END_METHOD

METHOD PROTECTED Internal_Insert
VAR_INPUT
	Data 		: T_Generic; // Data to insert
END_VAR
VAR_OUTPUT
	bSuccess 	: BOOL; // Indicates whether operation was successful. Success = TRUE, Failure = FALSE
END_VAR
VAR
	nState 		: DINT;
	pNew_Node,
	pCurrent	: POINTER TO T_BST_Node;
END_VAR
pNew_Node := THIS^.Malloc_Node(Data);

IF THIS^.pRoot = 0 THEN THIS^.pRoot := pNew_Node; bSuccess := TRUE; THIS^.IncrementCount(); RETURN; END_IF

pCurrent := THIS^.pRoot;
WHILE pCurrent <> 0 DO
	nState := THIS^.Compare(Data, pCurrent^.Data);
	CASE nState OF
	-1: // Less than
		IF pCurrent^.pLeft = 0 THEN pCurrent^.pLeft  := pNew_Node; bSuccess := TRUE; THIS^.IncrementCount(); RETURN; END_IF
		pCurrent  := pCurrent^.pLeft;
	 1: // Greater than
		IF pCurrent^.pRight = 0 THEN pCurrent^.pRight := pNew_Node; bSuccess := TRUE; THIS^.IncrementCount(); RETURN; END_IF
		pCurrent := pCurrent^.pRight;
	ELSE
		__DELETE(pNew_Node^.Data.pValue);
		__DELETE(pNew_Node);
		EXIT;
	END_CASE
	END_WHILE
END_METHOD

METHOD PROTECTED Internal_Remove : POINTER TO T_BST_Node
VAR_INPUT
	Data 		: T_Generic; // Data to remove
END_VAR
VAR_OUTPUT
	bSuccess 	: BOOL; 		// Indicates whether operation was successful. Success = TRUE, Failure = FALSE
END_VAR
VAR
	nState, nFirst 	: DINT;
	pCurrent, 
	pParent,
	pChild,
	pMin			: POINTER TO T_BST_Node;
	bInit 			: BOOL := TRUE;
END_VAR
pCurrent := THIS^.pRoot;
WHILE pCurrent <> 0 DO
	nState := THIS^.Compare(Data, pCurrent^.Data);
	IF bInit THEN nFirst := nState; bInit := FALSE; END_IF
	CASE nState OF
	 0: // Equal
	 	EXIT;
	-1: // Less than
		pParent := pCurrent; pCurrent := pCurrent^.pLeft;
	 1: // Greater than   
	 	pParent := pCurrent; pCurrent := pCurrent^.pRight;
	END_CASE
	END_WHILE

IF pCurrent = 0 THEN RETURN; END_IF // Return if node not found

bSuccess := TRUE;
THIS^.DecrementCount();
 
IF (pCurrent^.pLeft = 0) OR (pCurrent^.pRight = 0) THEN
	
	pChild := SEL(pCurrent^.pLeft = 0, pCurrent^.pLeft, pCurrent^.pRight);
	
	IF pParent = 0 				 THEN THIS^.pRoot := pChild; __DELETE(pCurrent^.Data.pValue); __DELETE(pCurrent);	  RETURN; END_IF	
	IF pCurrent = pParent^.pLeft THEN pParent^.pLeft := pChild;  __DELETE(pCurrent^.Data.pValue); __DELETE(pCurrent); RETURN; END_IF
	pParent^.pRight := pChild;  __DELETE(pCurrent^.Data.pValue); __DELETE(pCurrent); RETURN;
	END_IF 
	
pParent := pCurrent;
pMin 	:= pCurrent^.pRight;
WHILE (pMin^.pLeft <> 0) DO pParent := pMin; pMin := pMin^.pLeft; END_WHILE

pCurrent^.Data := pMin^.Data;
IF pMin = pParent^.pLeft THEN pParent^.pLeft := pMin^.pRight; ELSE pParent^.pRight := pMin^.pRight; END_IF
	
__DELETE(pMin^.Data.pValue);
__DELETE(pMin);
END_METHOD

// Checks if BST is Balanced
METHOD PROTECTED Is_Balanced : BOOL
END_METHOD

METHOD PROTECTED Malloc_Node : POINTER TO T_BST_Node
VAR_INPUT
	Data 	: T_Generic;
END_VAR
VAR
	pTemp 	: POINTER TO T_BST_Node;
END_VAR
pTemp 					:= __NEW(BYTE, SIZEOF(T_BST_Node));
pTemp^.Data.TypeClass 	:= Data.TypeClass;
pTemp^.Data.diSize 		:= Data.diSize;
pTemp^.Data.pValue 		:= __NEW(BYTE, TO_UDINT(Data.diSize));
MEMMOVE(pTemp^.Data.pValue, Data.pValue, TO_UDINT(Data.diSize));
Malloc_Node 			:= pTemp;
END_METHOD

// Gets the type of the data on the binary search tree
PROPERTY _Type : T_Type
GET
_Type := THIS^.Type_;
END_GET
SET
PROTECTED 
VAR
END_VAR
THIS^.Type_ := _Type;
END_SET
END_PROPERTY

// Balances Binary Search Tree. Tree will normal auto balance every time its count is a multiple of 4
METHOD Balance
VAR
	pTemp 			 	 : POINTER TO T_BST_Node;
	pStack 				 : POINTER TO FB_Stack;
	pStack_List,
	pOrdered_List 		 : POINTER TO FB_List;
	pHelper_BST_Balancer : POINTER TO FB_Helper_BST_Balancer;
END_VAR
IF THIS^.pRoot = 0 THEN RETURN; END_IF

// Create helpers
pHelper_BST_Balancer := __NEW(FB_Helper_BST_Balancer);
pStack_List 		 := __NEW(FB_List);
pOrdered_List 		 := __NEW(FB_List);
pStack 				 := __NEW(FB_Stack);
pStack^(ipList := pStack_List^);

// Inorder traversal
pTemp := THIS^.pRoot;
WHILE (pTemp <> 0) OR (NOT pStack^._Is_Empty) DO
	IF pTemp <> 0 THEN pStack^.Push(pTemp); pTemp := pTemp^.pLeft; CONTINUE; END_IF
	pStack^.Pop(pTemp); 
	pOrdered_List^.Add_Back(pTemp);
	pTemp := pTemp^.pRight;
	END_WHILE

// Balance BST
pTemp := 0;
pHelper_BST_Balancer^(ipList := pOrdered_List^, nStart := 0, nEnd := pOrdered_List^._Count -1 , pNode => pTemp);
IF pTemp <> 0 THEN THIS^.pRoot := pTemp; END_IF

// Delete helpers
__DELETE(pHelper_BST_Balancer);
__DELETE(pStack_List);
__DELETE(pStack);
__DELETE(pOrdered_List);











(*
pCurrent := THIS^.pRoot;
WHILE pCurrent <> 0 DO 
	IF pCurrent^.pLeft = 0 THEN pCurrent := pCurrent^.pRight;  CONTINUE; END_IF
	
	pPrevious := pCurrent^.pLeft;
	WHILE (pPrevious^.pRight <> 0 ) AND (pPrevious^.pRight <> pCurrent) DO
		pPrevious := pPrevious^.pRight;
		IF pPrevious^.pRight = 0 THEN pPrevious^.pRight := pCurrent; pCurrent := pCurrent^.pLeft; CONTINUE; END_IF
		pPrevious^.pRight := 0;
		pCurrent := pCurrent^.pRight;
		END_WHILE
	
	END_WHILE
*)
END_METHOD

(* Empties/Clears/Deletes every element on the collection *)
METHOD Clear
VAR
	pList 	: POINTER TO FB_List;
	pQueue 	: POINTER TO FB_Queue;
	pTemp 	: POINTER TO T_BST_Node;
END_VAR
IF THIS^.pRoot = 0 THEN RETURN; END_IF
pList 	:= __NEW(FB_List);
pQueue 	:= __NEW(FB_Queue);
pQueue^(ipList := pList^);

pQueue^.Enqueue(THIS^.pRoot);
WHILE NOT pQueue^._Is_Empty DO
	pQueue^.Dequeue(pTemp);
	IF pTemp^.pLeft <> 0 THEN pQueue^.Enqueue(pTemp^.pLeft);END_IF
	IF pTemp^.pRight <> 0 THEN pQueue^.Enqueue(pTemp^.pRight);END_IF
	
	__DELETE(pTemp^.Data.pValue);
	__DELETE(pTemp);
	THIS^.DecrementCount();
	END_WHILE

THIS^.pRoot := 0;
__DELETE(pQueue);
__DELETE(pList);
END_METHOD

METHOD FB_exit : BOOL
VAR_INPUT
	bInCopyCode : BOOL; // if TRUE, the exit method is called for exiting an instance that is copied afterwards (online change).
END_VAR
THIS^.Clear();
END_METHOD

METHOD FB_init : BOOL
VAR_INPUT
	bInitRetains 	: BOOL; // if TRUE, the retain variables are initialized (warm start / cold start)
	bInCopyCode 	: BOOL;  // if TRUE, the instance afterwards gets moved into the copy code (online change)
	eType 			: T_Type;
END_VAR
THIS^._Type := eType;
END_METHOD

(* Checks if data is contained in binary search tree *)
METHOD Find : I_Binary_Search_Tree
VAR_INPUT
	Data 		: ANY; 	// Data to remove
END_VAR
VAR_OUTPUT
	bFound 		: BOOL; // Indicates whether data was found. Found = TRUE, Not Found = FALSE
END_VAR
Find := THIS^;
IF THIS^.InvalidTypeException(Data) THEN RETURN; END_IF
THIS^.Internal_Find(Data, bFound => bFound);
END_METHOD

// Checks if generic data is inside binary search tree
METHOD Find_Generic : I_Generic_Binary_Search_Tree
VAR_INPUT
	Data 		: T_Generic; 	// Generic Data to find
END_VAR
VAR_OUTPUT
	bFound 		: BOOL; // Indicates whether data was found. Found = TRUE, Not Found = FALSE
END_VAR
Find_Generic := THIS^;
IF THIS^.InvalidTypeException(Data) THEN RETURN; END_IF
THIS^.Internal_Find(Data, bFound => bFound);
END_METHOD

(* Insert data into binary search tree *)
METHOD Insert : I_Binary_Search_Tree
VAR_INPUT
	Data 		: ANY; // Data to insert
END_VAR
VAR_OUTPUT
	bSuccess 	: BOOL; // Indicates whether operation was successful. Success = TRUE, Failure = FALSE
END_VAR
Insert := THIS^;
IF THIS^.InvalidTypeException(Data) THEN RETURN; END_IF
THIS^.Internal_Insert(Data, bSuccess => bSuccess);
IF (NOT THIS^.Balance_Ready()) OR (NOT bSuccess) THEN RETURN; END_IF
THIS^.Balance();
END_METHOD

// Adds new generic item at into binary search tree.
// The binary seach tree will store a copy of the generic item so as to not modify the original value outside it's scope.
METHOD Insert_Generic : I_Generic_Binary_Search_Tree
VAR_INPUT
	Data 	: T_Generic; // Item to store
END_VAR
VAR_OUTPUT
	bSuccess 	: BOOL; // Indicates whether operation was successful. Success = TRUE, Failure = FALSE
END_VAR
Insert_Generic := THIS^;
IF THIS^.InvalidTypeException(Data) THEN RETURN; END_IF
THIS^.Internal_Insert(Data, bSuccess => bSuccess);
IF (NOT THIS^.Balance_Ready()) OR (NOT bSuccess) THEN RETURN; END_IF
THIS^.Balance();
END_METHOD

(* Removes data from binary search tree *)
METHOD Remove : I_Binary_Search_Tree
VAR_INPUT
	Data : ANY; // Data to remove
END_VAR
VAR_OUTPUT
	bSuccess 	: BOOL; // Indicates whether operation was successful. Success = TRUE, Failure = FALSE
END_VAR
VAR
	nState 		: DINT;
	pCurrent, 
	pParent,
	pChild,
	pMin		: POINTER TO T_BST_Node;
END_VAR
Remove := THIS^;
IF THIS^.InvalidTypeException(Data) THEN RETURN; END_IF
THIS^.Internal_Remove(Data, bSuccess => bSuccess);
IF (NOT THIS^.Balance_Ready()) OR (NOT bSuccess) THEN RETURN; END_IF
THIS^.Balance();
END_METHOD

(* Traveses the binary search tree and appends into a collection *)
METHOD Traverse : I_Binary_Search_Tree
VAR_INPUT
	eMethod 		: T_BST_Traversal; // Method to traverse the binary search tree
	ipGeneric_List 	: I_Generic_List; 		// Collection to append data to.
END_VAR
VAR
	pList 		: POINTER TO FB_List;
	pQueue 		: POINTER TO FB_Queue;
	pStack 		: POINTER TO FB_Stack;
	pCurrent,
	pPrevious 	: POINTER TO T_BST_Node;
END_VAR
Traverse := THIS^;
IF THIS^.pRoot = 0 THEN RETURN; END_IF
IF ipGeneric_List = 0 THEN RETURN; END_IF

pList := __NEW(FB_List);

CASE eMethod OF
	T_BST_Traversal.Inorder:
		// In Order Traversal
		pStack := __NEW(FB_Stack);
		pStack^(ipList := pList^);
		pCurrent := THIS^.pRoot;
		WHILE (pCurrent <> 0) OR (NOT pStack^._Is_Empty) DO
			IF pCurrent <> 0 THEN pStack^.Push(pCurrent); pCurrent := pCurrent^.pLeft; CONTINUE; END_IF
			pStack^.Pop(pCurrent); 
			ipGeneric_List.Insert_Generic(pCurrent^.Data, ipGeneric_List._Count);
			pCurrent := pCurrent^.pRight;
			END_WHILE
		__DELETE(pStack);
		
	T_BST_Traversal.Postorder:
		// Post Order
		pStack := __NEW(FB_Stack);
		pStack^(ipList := pList^);
		pCurrent := THIS^.pRoot;
		
		WHILE (pCurrent <> 0) OR (NOT pStack^._Is_Empty) DO
			IF pCurrent <> 0 THEN pStack ^.Push(pCurrent); pCurrent := pCurrent^.pLeft; CONTINUE; END_IF
			pStack^.Top(pCurrent);
			IF (pCurrent^.pRight = 0) OR (pCurrent^.pRight = pPrevious) THEN 
				ipGeneric_List.Insert_Generic(pCurrent^.Data, ipGeneric_List._Count);
				pStack^.Pop_Void();
				pPrevious := pCurrent;
				pCurrent := 0;
				CONTINUE;
				END_IF
			pCurrent := pCurrent^.pRight;
			END_WHILE
		__DELETE(pStack);
		
	T_BST_Traversal.Preorder:
		// Preoder Traversal
		pStack := __NEW(FB_Stack);
		pStack^(ipList := pList^);
		pCurrent := THIS^.pRoot;
		pStack^.Push(pCurrent);
		WHILE NOT pStack^._Is_Empty DO
			pStack^.Pop(pCurrent);
			ipGeneric_List.Insert_Generic(pCurrent^.Data, ipGeneric_List._Count);
			IF pCurrent^.pRight <> 0 THEN pStack^.Push(pCurrent^.pRight); END_IF
			IF pCurrent^.pLeft  <> 0 THEN pStack^.Push(pCurrent^.pLeft); END_IF
			END_WHILE
		__DELETE(pStack);
		
	T_BST_Traversal.Level_Order:
		// Level Traversal
		pQueue 	:= __NEW(FB_Queue);
		pQueue^(ipList := pList^);
		pQueue^.Enqueue(THIS^.pRoot);
		WHILE NOT pQueue^._Is_Empty DO
			pQueue^.Dequeue(pCurrent);
			IF pCurrent^.pLeft <> 0 THEN pQueue^.Enqueue(pCurrent^.pLeft);END_IF
			IF pCurrent^.pRight <> 0 THEN pQueue^.Enqueue(pCurrent^.pRight);END_IF
			ipGeneric_List.Insert_Generic(pCurrent^.Data, ipGeneric_List._Count);
			END_WHILE
		__DELETE(pQueue);
END_CASE
__DELETE(pList);
END_METHOD

END_FUNCTION_BLOCK

// POUs/Function Blocks/Helpers/FB_Helper_BST_Balancer
// Helper to balance Binary Search Tree since recurssion is not supported
{attribute 'enable_dynamic_creation'}
FUNCTION_BLOCK INTERNAL FINAL FB_Helper_BST_Balancer
VAR_INPUT
	ipList 			: I_List;
	nStart,
	nEnd 			: T_Capacity;  
END_VAR
VAR_OUTPUT
	pNode 			: POINTER TO T_BST_Node;
END_VAR
VAR
	bSuccess		: BOOL;
	nMid 			: T_Capacity;
	pTree_Balancer 	: POINTER TO FB_Helper_BST_Balancer;
END_VAR

IF ipList = 0 THEN RETURN; END_IF
IF nStart > nEnd THEN RETURN; END_IF

nMid := (nStart+nEnd)/2;
ipList.Get(pNode, nMid, bSuccess => bSuccess);
IF (NOT bSuccess) OR pNode = 0 THEN RETURN; END_IF 

pTree_Balancer := __NEW(FB_Helper_BST_Balancer);
pTree_Balancer^(ipList := ipList, nStart := nStart, nEnd := nMid-1, pNode => pNode^.pLeft);
pTree_Balancer^(ipList := ipList, nStart := nMid+1, nEnd := nEnd, 	pNode => pNode^.pRight);
__DELETE(pTree_Balancer);

END_FUNCTION_BLOCK

// POUs/Function Blocks/FB_List
// Dyanamic List that can store a collection of any types. Similiar to python lists.
{attribute 'enable_dynamic_creation'}
{attribute 'no_assign'}
FUNCTION_BLOCK FB_List EXTENDS FB_Collection IMPLEMENTS I_List, I_Generic_List
VAR
	pHead, pTail	: POINTER TO ST_LIST_NODE;
END_VAR

// Raises an expection if list is empty
METHOD PROTECTED EmptyListException : BOOL
VAR_INPUT
END_VAR
IF THIS^._Is_Empty THEN
	stError.bSTATUS := TRUE;
	stError.nCODE 	:= 2936;
	stError.sSOURCE := 'List is empty';
ELSE
	This^.ClearException();
	END_IF
EmptyListException := stError.bSTATUS;
END_METHOD

// Compares memory sizes of 2 addresses. Returns TRUE  and raises error flag if theyre not same size.
METHOD PROTECTED MemCmpErrExpection : BOOL
VAR_INPUT
	pDestAddr,
	pSrcAddr 	: PVOID;
	nSize 		: UDINT;
END_VAR
VAR_INST
	nMemErr : DINT;
END_VAR
nMemErr := MEMCMP(pDestAddr, pSrcAddr, nSize);
IF nMemErr = -1 THEN 
	stError.bSTATUS := TRUE;
	stError.nCODE 	:= 4129;
	stError.sSOURCE := 'Incorrect parameter values. Destination address smaller than source address';
	
ELSIF nMemErr = 0 THEN THIS^.ClearException();
	
ELSIF nMemErr = 1 THEN
	stError.bSTATUS := TRUE;
	stError.nCODE 	:= 4823;
	stError.sSOURCE := 'Incorrect parameter values. Destination address greater that source address';

ELSE
	stError.bSTATUS := TRUE;
	stError.nCODE 	:= 4564;
	stError.sSOURCE := 'Incorrect parameter values. Pointer to destination/source address is NULL or allocated address memory is NULL.';
	END_IF

MemCmpErrExpection := stError.bSTATUS;
END_METHOD

METHOD PROTECTED OutOfBoundsException : BOOL
VAR_INPUT
	nIndex : DINT;
END_VAR
IF (nIndex < 0) OR (nIndex >= THIS^._Count) THEN
	stError.bSTATUS := TRUE;
	stError.nCODE 	:= 5374;
	stError.sSOURCE := 'Out of bounds. You tried to access data outside the range of this list.';
ELSE
	This^.ClearException();
	END_IF
OutOfBoundsException := stError.bSTATUS;
END_METHOD

METHOD TypeMismatchException : BOOL
VAR_INPUT
	Dest,
	Src 	: __SYSTEM.AnyType;
END_VAR
IF Dest.diSize <> Src.diSize THEN
	stError.bSTATUS := TRUE;
	stError.nCODE 	:= 3172;
	stError.sSOURCE := 'Type mismatch. Byte sizes are not the same';
ELSIF Dest.TypeClass <> Src.TypeClass THEN
	stError.bSTATUS := TRUE;
	stError.nCODE 	:= 3172;
	stError.sSOURCE := 'Type mismatch. Type classes are not the same';
ELSE
	THIS^.ClearException();
END_IF
TypeMismatchException := stError.bSTATUS;
END_METHOD

// Copy data from source memory space to desination memory space
METHOD PROTECTED CopyValueTo
VAR_INPUT
	Dest, Src : __SYSTEM.AnyType;
END_VAR
MEMMOVE(Dest.pValue, Src.pValue, TO_UDINT(Dest.diSize));
END_METHOD

// Decrement list size by 1.
METHOD PROTECTED DecrementCount
VAR_INPUT
END_VAR
THIS^.nCount := THIS^.nCount - 1;
END_METHOD

// Deletes/frees node and it's value from memory
METHOD PROTECTED Free_Node
VAR_INPUT
	pNode : POINTER TO ST_LIST_NODE; 
END_VAR
IF pNode^.Data.pValue <> 0 THEN  __DELETE(pNode^.Data.pValue); END_IF
IF pNode <> 0 THEN __DELETE(pNode); END_IF
END_METHOD

METHOD PROTECTED GetValueAsString : T_MaxString
VAR_INPUT
	 Value : __SYSTEM.AnyType;
END_VAR
VAR	
	pBool			: POINTER TO BOOL;
    pByte			: POINTER TO BYTE;
    pWord			: POINTER TO WORD;
    pDWord			: POINTER TO DWORD;
    pLWord			: POINTER TO LWORD;
    pSint			: POINTER TO SINT;
    pInt			: POINTER TO INT;
    pDint			: POINTER TO DINT;
    pLint			: POINTER TO LINT;
    pUSint			: POINTER TO USINT;
    pUInt			: POINTER TO UINT;
    pUDint			: POINTER TO UDINT;
    pULint			: POINTER TO ULINT;
    pReal			: POINTER TO REAL;
    pLReal			: POINTER TO LREAL;
    pString			: POINTER TO STRING(255);
    pWString		: POINTER TO WSTRING;
    pTime			: POINTER TO TIME;
    pDate			: POINTER TO DATE;
    pDate_And_Time	: POINTER TO DATE_AND_TIME;
    pTime_Of_Day	: POINTER TO TIME_OF_DAY;
    pPointer		: PVOID;
	pLTime 			: POINTER TO LTIME;
END_VAR
IF Value.pValue = 0 THEN GetValueAsString := 'NULL'; RETURN; END_IF;

CASE Value.TypeClass OF 
	__SYSTEM.TYPE_CLASS.TYPE_BOOL:
		pBool := Value.pValue;
		GetValueAsString := TO_STRING(pBool^);
		
    __SYSTEM.TYPE_CLASS.TYPE_BYTE:
		pByte := Value.pValue;
		GetValueAsString := TO_STRING(pByte^);
		
    __SYSTEM.TYPE_CLASS.TYPE_WORD:
		pWord := Value.pValue;
		GetValueAsString := TO_STRING(pWord^);
		
    __SYSTEM.TYPE_CLASS.TYPE_DWORD:
		pDWord := Value.pValue;
		GetValueAsString := TO_STRING(pDWord^);
		
    __SYSTEM.TYPE_CLASS.TYPE_LWORD:
		pLWord := Value.pValue;
		GetValueAsString := TO_STRING(pLWord^);
		
    __SYSTEM.TYPE_CLASS.TYPE_SINT:
		pSint := Value.pValue;
		GetValueAsString := TO_STRING(pSint^);
		
    __SYSTEM.TYPE_CLASS.TYPE_INT:
		pInt := Value.pValue;
		GetValueAsString := TO_STRING(pInt^);
		
    __SYSTEM.TYPE_CLASS.TYPE_DINT:
		pDint := Value.pValue;
		GetValueAsString := TO_STRING(pDint^);
		
    __SYSTEM.TYPE_CLASS.TYPE_LINT:
		pLint := Value.pValue;
		GetValueAsString := TO_STRING(pLint^);
		
    __SYSTEM.TYPE_CLASS.TYPE_USINT:
		pUSint := Value.pValue;
		GetValueAsString := TO_STRING(pUSint^);
		
    __SYSTEM.TYPE_CLASS.TYPE_UINT:
		pUInt := Value.pValue;
		GetValueAsString := TO_STRING(pUInt^);
		
    __SYSTEM.TYPE_CLASS.TYPE_UDINT:
		pUDint := Value.pValue;
		GetValueAsString := TO_STRING(pUDint^);
		
    __SYSTEM.TYPE_CLASS.TYPE_ULINT:
		pULint := Value.pValue;
		GetValueAsString := TO_STRING(pULint^);
		
   __SYSTEM.TYPE_CLASS.TYPE_REAL:
		pReal := Value.pValue;
		GetValueAsString := TO_STRING(pReal^);
		
    __SYSTEM.TYPE_CLASS.TYPE_LREAL:
		pLReal := Value.pValue;
		GetValueAsString := TO_STRING(pLReal^);
		
    __SYSTEM.TYPE_CLASS.TYPE_STRING:
		pString := Value.pValue;
		GetValueAsString := TO_STRING(pString^);
		
   __SYSTEM.TYPE_CLASS.TYPE_WSTRING:
		pWString := Value.pValue;
		GetValueAsString := TO_STRING(pWString^);
		
    __SYSTEM.TYPE_CLASS.TYPE_TIME:
		pTime := Value.pValue;
		GetValueAsString := TO_STRING(pTime^);
		
    __SYSTEM.TYPE_CLASS.TYPE_DATE:
		pDate := Value.pValue;
		GetValueAsString := TO_STRING(pDate^);
		
    __SYSTEM.TYPE_CLASS.TYPE_DATEANDTIME:
		pDate_And_Time := Value.pValue;
		GetValueAsString := TO_STRING(pDate_And_Time^);
		
    __SYSTEM.TYPE_CLASS.TYPE_TIMEOFDAY:
		pTime_Of_Day := Value.pValue;
		GetValueAsString := TO_STRING(pTime_Of_Day^);
	
	__SYSTEM.TYPE_CLASS.TYPE_POINTER:
		GetValueAsString := TO_STRING(Value.pValue);
		
	__SYSTEM.TYPE_CLASS.TYPE_LTIME:
		pLTime := Value.pValue;
		GetValueAsString := TO_STRING(pLTime^);
ELSE
	GetValueAsString := 'TYPE TO STRING CONVERSION NOT SUPPORTED BY THIS TYPE'; 
END_CASE
END_METHOD

// Increments list size by 1
METHOD PROTECTED IncrementCount
VAR_INPUT
END_VAR
THIS^.nCount := THIS^.nCount + 1;
END_METHOD

// Returns pointer to node at specificied location;
METHOD PROTECTED Iterate : POINTER TO ST_LIST_NODE
VAR_INPUT
	nIndex : T_Capacity;
END_VAR
VAR_INST
	nState : BYTE;
	ii : T_Capacity;
	pT : POINTER TO ST_LIST_NODE;
END_VAR
VAR 
	i 		: DINT;
	pTemp 	: POINTER TO ST_LIST_NODE;
END_VAR
IF THIS^.OutOfBoundsException(nIndex) THEN RETURN; END_IF
IF nIndex = 0 THEN Iterate := THIS^.pHead; RETURN; END_IF
//IF nIndex = THIS^._Count - 1 THEN Iterate := pTail; RETURN; END_IF {warning 'changes made here'}
pTemp := pHead;
FOR i := 1 TO nIndex DO pTemp := pTemp^.pNext; END_FOR
Iterate := pTemp;
END_METHOD

// Allocate memory space for node and the value for it's data on the heap, returns pointer to node;
// WARNING!!! Always have a place to store the node pointer otherwise a memory leak will occur.
METHOD PROTECTED Malloc_Node : POINTER TO ST_LIST_NODE
VAR_INPUT
	Variable : __SYSTEM.AnyType;
END_VAR
VAR
	pTemp 	: POINTER TO ST_LIST_NODE;
END_VAR
pTemp 					:= __NEW(ST_LIST_NODE); // Allocate space in memory for a node.
pTemp^.Data.sValue 		:= THIS^.GetValueAsString(Variable);
pTemp^.Data.pValue 		:= __NEW(BYTE, TO_UDINT(Variable.diSize)); // Allocate space in memory to store data value.
pTemp^.Data.diSize 		:= Variable.diSize;
pTemp^.Data.TypeClass 	:= Variable.TypeClass;

Malloc_Node := pTemp;
END_METHOD

(* Set value of __SYSTEM.Anytype variable *)
METHOD PROTECTED SetValue
VAR_INPUT
	Variable	: __SYSTEM.Anytype;
	Value 		: USINT; // Character/byte to set.
END_VAR
MEMSET(Variable.pValue, Value, TO_UDINT(Variable.diSize));
END_METHOD

(* Checks of list is empty.*)
PROPERTY _Is_Empty : BOOL
GET
_Is_Empty := (THIS^._Count = 0);
END_GET
END_PROPERTY

// Adds an item to the end of the list
METHOD Add_Back : I_List
VAR_INPUT
	Item 	: ANY; // Value to store in list
END_VAR
VAR_OUTPUT
	bSuccess : BOOL;
END_VAR
VAR
	pTemp 	: POINTER TO ST_LIST_NODE;
END_VAR
Add_Back := THIS^;
IF THIS^._Is_Empty THEN THIS^.Add_Front(Item, bSuccess => bSuccess); RETURN; END_IF
pTemp := THIS^.Malloc_Node(Item);
THIS^.CopyValueTo(pTemp^.Data, Item);
THIS^.pTail := THIS^.pTail^.pNext := pTemp;
THIS^.IncrementCount();
END_METHOD

// Adds an item at the front of the list
METHOD Add_Front : I_List
VAR_INPUT
	Item 	: ANY; // Item to store in list
END_VAR
VAR_OUTPUT
	bSuccess : BOOL;
END_VAR
VAR
	pTemp 	: POINTER TO ST_LIST_NODE;
END_VAR
Add_Front := THIS^;
pTemp := THIS^.Malloc_Node(Item);
THIS^.CopyValueTo(pTemp^.Data, Item);
pTemp^.pNext := THIS^.pHead; THIS^.pHead := pTemp;
IF THIS^._Is_Empty THEN THIS^.pTail := THIS^.pHead; END_IF
THIS^.IncrementCount();
bSuccess := TRUE;
END_METHOD

(* Empties/Clears/Deletes every item in the list *)
METHOD Clear
VAR
	pTemp : POINTER TO ST_LIST_NODE;
END_VAR
pTemp := THIS^.pHead;
WHILE pTemp <> 0 DO
	pTemp := pTemp^.pNext; THIS^.Remove();
END_WHILE
END_METHOD

(* Checks if item is contained in list *)
METHOD Contains : BOOL
VAR_INPUT
	Item : ANY; // Item to find in list
END_VAR
VAR
	nIndex : DINT := -1;
END_VAR
THIS^.Find(Item, nIndex => nIndex, bSuccess => Contains);
END_METHOD

METHOD FB_exit : BOOL
VAR_INPUT
	(* if TRUE, the exit method is called for exiting an instance that is copied afterwards (online change).*)
	bInCopyCode	: BOOL;
END_VAR
This^.Clear();
END_METHOD

METHOD FB_init : BOOL
VAR_INPUT
	bInitRetains : BOOL; // if TRUE, the retain variables are initialized (warm start / cold start)
	bInCopyCode : BOOL;  // if TRUE, the instance afterwards gets moved into the copy code (online change)
END_VAR
THIS^.Clear();
THIS^.pHead := THIS^.pTail := Tc3_Module.GVL.NULL;
END_METHOD

// Find the location of an item in list.
METHOD Find : I_List
VAR_INPUT
	Item 	 : ANY; // Item to find in list
END_VAR
VAR_OUTPUT
	nIndex	 : T_Capacity; //Location of item in list 
	bSuccess : BOOL;
END_VAR
VAR
	pTemp 	 : POINTER TO ST_LIST_NODE;
	i 		 : DINT;
	n 		 : DINT := -1;
END_VAR
Find := THIS^;
IF THIS^.EmptyListException() THEN nIndex := -1; RETURN; END_IF
pTemp := THIS^.pHead;
FOR i := 0 TO THIS^._Count-1 DO
	IF pTemp = 0 THEN EXIT; END_IF
	IF (pTemp^.Data.pValue = 0) 					THEN pTemp := pTemp^.pNext; CONTINUE; END_IF
	IF (Item.TypeClass <> pTemp^.Data.TypeClass) 	THEN pTemp := pTemp^.pNext; CONTINUE; END_IF
	IF (Item.pValue^ <> pTemp^.Data.pValue^) 		THEN pTemp := pTemp^.pNext; CONTINUE; END_IF
	
	CASE Item.TypeClass OF
		__SYSTEM.TYPE_CLASS.TYPE_STRING:
			IF LEN2(Item.pValue) <> LEN2(pTemp^.Data.pValue) THEN pTemp := pTemp^.pNext; CONTINUE; END_IF
			n := MEMCMP(Item.pValue, pTemp^.Data.pValue, LEN2(pTemp^.Data.pValue)+1);
				
		__SYSTEM.TYPE_CLASS.TYPE_WSTRING:
			IF WLEN2(Item.pValue) <> WLEN2(pTemp^.Data.pValue) THEN pTemp := pTemp^.pNext; CONTINUE; END_IF
			n := MEMCMP(Item.pValue, pTemp^.Data.pValue, (WLEN2(pTemp^.Data.pValue)*SIZEOF(WORD))+1);
	ELSE
		IF (Item.diSize <> pTemp^.Data.diSize) THEN pTemp := pTemp^.pNext; CONTINUE; END_IF	
		n := MEMCMP(Item.pValue, pTemp^.Data.pValue, TO_UDINT(Item.diSize));
	END_CASE
	IF n = 0 THEN nIndex := i; bSuccess := TRUE; RETURN; END_IF
	pTemp := pTemp^.pNext;
	END_FOR
nIndex := -1;
END_METHOD

// Gets item from list at specified location without removing it
METHOD Get : I_List
VAR_INPUT
	Return_Item 	: ANY;  // Variable to store returned item
	nIndex 			: T_Capacity; // Location of item
END_VAR
VAR_OUTPUT
	bSuccess 		: BOOL;
END_VAR
VAR
	pTemp : POINTER TO ST_LIST_NODE;
END_VAR
Get := THIS^;
IF THIS^.EmptyListException() THEN RETURN; END_IF
IF THIS^.OutOfBoundsException(nIndex) THEN RETURN; END_IF
IF nIndex = 0 THEN THIS^.Get_First(Return_Item, bSuccess => bSuccess); RETURN; END_IF
IF nIndex = THIS^._Count - 1 THEN THIS^.Get_Last(Return_Item, bSuccess => bSuccess); RETURN; END_IF
pTemp := Iterate(nIndex);
IF THIS^.TypeMismatchException(Return_Item, pTemp^.Data) THEN RETURN; END_IF
THIS^.CopyValueTo(Return_Item, pTemp^.Data);
bSuccess := TRUE;
END_METHOD

// Gets item at the front of the list 
METHOD Get_First : I_List
VAR_INPUT
	Return_Item 	: ANY; // Variable to store returned item
END_VAR
VAR_OUTPUT
	bSuccess : BOOL;
END_VAR
Get_First := THIS^;
IF THIS^.EmptyListException() THEN RETURN; END_IF
IF THIS^.TypeMismatchException(Return_Item, pHead^.Data) THEN RETURN; END_IF
THIS^.CopyValueTo(Return_Item, pHead^.Data);
bSuccess := TRUE;
END_METHOD

// Gets a value from a collection in it's generic form (* Use carefully as this contains the pointer of the action value in the collection. *)
METHOD Get_Generic : I_Generic_List
VAR_INPUT
	nIndex 		: T_Capacity; 			// Location of item
END_VAR
VAR_OUTPUT
	Return_Item : T_Generic;  	// Variable to store returned item
	bSuccess 	: BOOL;
END_VAR
VAR
	pTemp : POINTER TO ST_LIST_NODE;
END_VAR
Get_Generic := THIS^;
IF THIS^.EmptyListException() THEN RETURN; END_IF
IF THIS^.OutOfBoundsException(nIndex) THEN RETURN; END_IF

IF nIndex = THIS^._Count - 1 THEN pTemp := pTail; ELSE pTemp := THIS^.Iterate(nIndex); END_IF
Return_Item := pTemp^.Data;
bSuccess := TRUE;
END_METHOD

// Gets item at the back of the list 
METHOD Get_Last : I_List
VAR_INPUT
	Return_Item 	: ANY; // Variable to store returned item
END_VAR
VAR_OUTPUT
	bSuccess : BOOL;
END_VAR
Get_Last := THIS^;
IF THIS^.EmptyListException() THEN RETURN; END_IF
IF THIS^.TypeMismatchException(Return_Item, pTail^.Data) THEN RETURN; END_IF
THIS^.CopyValueTo(Return_Item, pTail^.Data);
bSuccess := TRUE;
END_METHOD

// Returns item as a string, if type to string conversion is supported
METHOD Get_Value_As_String : I_List
VAR_INPUT
	nIndex	: T_Capacity; // Location of item
END_VAR
VAR_OUTPUT
	sItem 	: T_MaxString; // Variable to store returned item
END_VAR
VAR
	pTemp : POINTER TO ST_LIST_NODE;
END_VAR
Get_Value_As_String := THIS^;
IF THIS^.EmptyListException() OR THIS^.OutOfBoundsException(nIndex) THEN sItem := 'ERR: List is Empty or index Out of Bounds'; RETURN; END_IF
pTemp := Iterate(nIndex);
sItem := pTemp^.Data.sValue;
END_METHOD

// Adds new item to list at specified location, if index = 0, item will be added at the front, if index = count, item will be added at the back
METHOD Insert : I_List
VAR_INPUT
	Item 	: ANY;  // Item to store in list
	nIndex 	: T_Capacity; // Location of item
END_VAR
VAR_OUTPUT
	bSuccess : BOOL;
END_VAR
VAR
	pPrevious 	: POINTER TO ST_LIST_NODE;
	pCurrent 	: POINTER TO ST_LIST_NODE;
	pTemp 		: POINTER TO ST_LIST_NODE;
END_VAR
Insert := THIS^;
IF nIndex = 0 THEN THIS^.Add_Front(Item, bSuccess => bSuccess); RETURN; END_IF
IF nIndex = THIS^._Count THEN THIS^.Add_Back(Item, bSuccess => bSuccess); RETURN; END_IF
IF THIS^.OutOfBoundsException(nIndex) THEN RETURN; END_IF

pTemp := THIS^.Malloc_Node(Item);
THIS^.CopyValueTo(pTemp^.Data, Item);

pPrevious := THIS^.Iterate(nIndex-1);
pCurrent := pPrevious^.pNext;
pPrevious^.pNext := pTemp;
pTemp^.pNext := pCurrent;

THIS^.IncrementCount();
bSuccess := TRUE;
END_METHOD

// Adds new item to list at specified location using the generic form. If index = 0, item will be added at the front, if index = count, item will be added at the back
// To void race condition and memory leaks, a copy of the data/item in the generic form will be inserted. The original generic remains safe.
METHOD Insert_Generic : I_Generic_List
VAR_INPUT
	Item 	: T_Generic;  	// Item to store in list
	nIndex 	: T_Capacity; 			// Location of item
END_VAR
VAR_OUTPUT
	bSuccess : BOOL;
END_VAR
VAR
	pPrevious, pCurrent, pTemp : POINTER TO ST_LIST_NODE;
END_VAR
Insert_Generic := THIS^;

pTemp := THIS^.Malloc_Node(Item);
THIS^.CopyValueTo(pTemp^.Data, Item);

// Add to front if nIndex = 0
IF nIndex = 0 THEN
	pTemp^.pNext := THIS^.pHead; THIS^.pHead := pTemp;
	IF THIS^._Is_Empty THEN THIS^.pTail := THIS^.pHead; END_IF
	THIS^.IncrementCount();
	bSuccess := TRUE;
	RETURN; 
	END_IF
	
// Add to back if nIndex = Count
IF nIndex = THIS^._Count THEN 
	THIS^.pTail := THIS^.pTail^.pNext := pTemp;
	THIS^.IncrementCount();
	bSuccess := TRUE;
	RETURN;
	END_IF

// Free temp node and return if the node is out of bounds
IF THIS^.OutOfBoundsException(nIndex) THEN THIS^.Free_Node(pTemp); RETURN; END_IF

// Insert value at specified position position if all checks are passed
pPrevious := THIS^.Iterate(nIndex-1);
pCurrent := pPrevious^.pNext;
pPrevious^.pNext := pTemp;
pTemp^.pNext := pCurrent;

THIS^.IncrementCount();
bSuccess := TRUE;
END_METHOD

// Removes item at the front of the list and returns nothing
METHOD Remove : I_List
VAR_OUTPUT
	bSuccess : BOOL;
END_VAR
VAR
	pTemp 	: POINTER TO ST_LIST_NODE;
END_VAR
Remove := THIS^;
IF THIS^._Is_Empty THEN RETURN; END_IF

pTemp := THIS^.pHead^.pNext;
THIS^.Free_Node(pHead);
THIS^.pHead := pTemp;

IF THIS^._Count = 1 THEN pTail := 0; END_IF

THIS^.DecrementCount();
bSuccess := TRUE;
END_METHOD

// Remove item at specified location and return nothing
METHOD Remove_At : I_List
VAR_INPUT
	nIndex : T_Capacity; // Location of item
END_VAR
VAR_OUTPUT
	bSuccess : BOOL;
END_VAR
VAR
	pTemp : ARRAY[1..2] OF POINTER TO ST_LIST_NODE;
END_VAR
Remove_At := THIS^;
IF THIS^.EmptyListException() OR THIS^.OutOfBoundsException(nIndex) THEN RETURN; END_IF
IF nIndex = 0 THEN THIS^.Remove(bSuccess => bSuccess); RETURN; END_IF
IF nIndex = THIS^._Count - 1 THEN THIS^.Remove_Last(bSuccess => bSuccess); RETURN; END_IF

pTemp[1] := THIS^.Iterate(nIndex-1);
pTemp[2] := pTemp[1]^.pNext^.pNext;
THIS^.Free_Node(pTemp[1]^.pNext);
pTemp[1]^.pNext := pTemp[2];

THIS^.DecrementCount();
bSuccess := TRUE;
END_METHOD

// Removes item at the back of the list and returns nothing
METHOD Remove_Last : I_List
VAR_OUTPUT
	bSuccess : BOOL;
END_VAR
VAR
	pTemp : POINTER TO ST_LIST_NODE;
END_VAR
Remove_Last := THIS^;
IF THIS^.EmptyListException() THEN RETURN; END_IF
IF THIS^._Count = 1 THEN THIS^.Remove(bSuccess => bSuccess); RETURN; END_IF
pTemp := THIS^.Iterate(THIS^._Count - 2);
THIS^.Free_Node(pTemp^.pNext);
pTail := pTemp;
THIS^.DecrementCount();
bSuccess := TRUE;
END_METHOD

// Manually resize list. If list becomes smaller, items on higher locations will be deleted.
METHOD Resize : I_List
VAR_INPUT
	nSize : T_Capacity; // New size of list.
END_VAR
VAR_OUTPUT
	bSuccess : BOOL;
END_VAR
VAR 
	Data 		: __SYSTEM.AnyType;
	nCount,i	: DINT;
END_VAR
Resize := THIS^;
IF (nSize = THIS^._Count) OR (nSize < 0) THEN RETURN; END_IF 
IF nSize = 0 THEN THIS^.Clear(); bSuccess := TRUE; END_IF

nCount := THIS^._Count;

IF nSize < THIS^._Count THEN
	FOR i := 0 TO nCount - 1 DO
		THIS^.Remove_At(nCount - 1 - i, bSuccess => bSuccess);
		IF THIS^._Count = nSize THEN RETURN; END_IF
		END_FOR
	END_IF
	
IF nSize > THIS^._Count THEN
	FOR i := nCount TO nSize - 1 DO
		THIS^.Add_Back(Data, bSuccess => bSuccess);
		END_FOR
	END_IF
	
bSuccess := TRUE;
END_METHOD

// Reverses the order of items in the list
METHOD Reverse : I_List
VAR_OUTPUT
	bSuccess : BOOL;
END_VAR
VAR
	pPrevious 	: POINTER TO ST_LIST_NODE;
	pCurrent 	: POINTER TO ST_LIST_NODE;
	pNext	 	: POINTER TO ST_LIST_NODE;
END_VAR
Reverse := THIS^;
IF THIS^._Count = 1 OR THIS^.EmptyListException() THEN RETURN; END_IF
pCurrent := THIS^.pTail := THIS^.pHead;
WHILE pCurrent <> 0 DO
	pNext := pCurrent^.pNext;
	pCurrent^.pNext := pPrevious;
	pPrevious := pCurrent;
	pCurrent := pNext;
	END_WHILE
THIS^.pHead := pPrevious;
bSuccess := TRUE;
END_METHOD

// Adds new item to list in the specified location without resizing list
METHOD Set : I_List
VAR_INPUT
	Item 	: ANY; 	// Item to store in list
	nIndex 	: T_Capacity; // Location of item
END_VAR
VAR_OUTPUT
	bSuccess : BOOL;
END_VAR
VAR
	pTemp : POINTER TO ST_LIST_NODE;
END_VAR
Set := THIS^;
IF THIS^.OutOfBoundsException(nIndex) THEN RETURN; END_IF

IF nIndex = THIS^._Count - 1 THEN 
	pTemp := THIS^.pTail;
ELSE 
	pTemp := Iterate(nIndex);
	END_IF

__DELETE(pTemp^.Data.pValue); 

pTemp^.Data.sValue 		:= THIS^.GetValueAsString(Item);
pTemp^.Data.pValue 		:= __NEW(BYTE, TO_UDINT(Item.diSize)); // Allocate space in memory to store data value.
pTemp^.Data.diSize 		:= Item.diSize;
pTemp^.Data.TypeClass 	:= Item.TypeClass;

THIS^.CopyValueTo(pTemp^.Data, Item);
bSuccess := TRUE;
END_METHOD

END_FUNCTION_BLOCK

// POUs/Function Blocks/FB_Stack
{attribute 'enable_dynamic_creation'}
{attribute 'no_assign'}
FUNCTION_BLOCK FB_Stack EXTENDS FB_Collection IMPLEMENTS I_Stack
VAR_INPUT
	ipList : I_List; // List to perform operations on.
END_VAR
VAR_OUTPUT
END_VAR

METHOD PROTECTED NullReferenceException : BOOL
NullReferenceException := THIS^.ipList = 0;
IF NOT NullReferenceException THEN RETURN; END_IF
THIS^.RaiseException(2000+GVL_CmpErrors.ERR_INVALID_REFERENCE, 'Null or Invalid Reference');
END_METHOD

METHOD PROTECTED CatchError : BOOL
VAR_INPUT
END_VAR
stError := THIS^.ipList._Error_Status;
CatchError := stError.bSTATUS;
END_METHOD

(* Number of elements in the stack *)
PROPERTY _Count : T_Capacity
GET
IF THIS^.NullReferenceException() THEN _Count := -1; RETURN; END_IF
_Count := THIS^.ipList._Count;
END_GET
END_PROPERTY

PROPERTY _Error_Status : ST_ERROR
GET
IF THIS^.NullReferenceException() THEN _Error_Status := THIS^.stError; RETURN; END_IF
THIS^.stError := THIS^.ipList._Error_Status;
_Error_Status := F_Error(THIS^.stError.bSTATUS, THIS^.stError.nCODE, THIS^.stError.sSOURCE);
END_GET
END_PROPERTY

(* Checks of stack is empty.*)
PROPERTY _Is_Empty : BOOL
GET
IF THIS^.NullReferenceException() THEN _Is_Empty := TRUE; RETURN; END_IF
_Is_Empty := THIS^.ipList._Is_Empty;
END_GET
END_PROPERTY

(* Empties/Clears/Deletes every item on the stack*)
METHOD Clear
VAR_INPUT
END_VAR
IF THIS^.NullReferenceException() THEN RETURN; END_IF
THIS^.ipList.Clear();
END_METHOD

(* Get item from stack without removing it. *)
METHOD Peek : I_Stack
VAR_INPUT
	Item 	: ANY; (* Variable to store returned item value *)
	nIndex 	: DINT; (* Location of item*)
END_VAR
VAR_OUTPUT
	bSuccess : BOOL;
END_VAR
Peek := THIS^;
IF THIS^.NullReferenceException() THEN RETURN; END_IF
THIS^.ipList.Get(Item, nIndex, bSuccess => bSuccess);
END_METHOD

(* Gets and deletes item at the top of the stack *)
METHOD Pop : I_Stack
VAR_INPUT
	Item : ANY; (* Variable to store returned item value *)
END_VAR
VAR_OUTPUT
	bSuccess : BOOL;
END_VAR
VAR
	bA, bB 	 : BOOL;
END_VAR
Pop := THIS^;
IF THIS^.NullReferenceException() THEN RETURN; END_IF
THIS^.ipList.Get_First(Item, bSuccess => bA).Remove( bSuccess => bB);
bSuccess := bA AND bB;
END_METHOD

(* Removes item at the top of the stack without returning anything *)
METHOD Pop_Void : I_Stack
VAR_OUTPUT
	bSuccess : BOOL;
END_VAR
Pop_Void := THIS^;
IF THIS^.NullReferenceException() THEN RETURN; END_IF
THIS^.ipList.Remove(bSuccess => bSuccess);
END_METHOD

(* Add item to the top of the stack *)
METHOD Push : I_Stack
VAR_INPUT
	Item : ANY; (* Variable containg data to store on the stack *)
END_VAR
VAR_OUTPUT
	bSuccess : BOOL;
END_VAR
Push := THIS^;
IF THIS^.NullReferenceException() THEN RETURN; END_IF
THIS^.ipList.Add_Front(Item, bSuccess => bSuccess);
END_METHOD

(* Reverses order of items on stack *)
METHOD Reverse : I_Stack
VAR_OUTPUT
	bSuccess : BOOL;
END_VAR
Reverse := THIS^;
IF THIS^.NullReferenceException() THEN RETURN; END_IF
THIS^.ipList.Reverse(bSuccess => bSuccess);
END_METHOD

(* Get item at the top of the stack without removing it. *)
METHOD Top : I_Stack
VAR_INPUT
	Item 	: ANY; (* Variable to store returned item value *)
END_VAR
VAR_OUTPUT
	bSuccess : BOOL;
END_VAR
Top := THIS^;
IF THIS^.NullReferenceException() THEN RETURN; END_IF
THIS^.ipList.Get_First(Item, bSuccess => bSuccess);
END_METHOD

END_FUNCTION_BLOCK

// POUs/Function Blocks/FB_Queue
// Queue Decorator for function blocks that impliment I_List interface
{attribute 'enable_dynamic_creation'}
FUNCTION_BLOCK FB_Queue EXTENDS FB_Collection  IMPLEMENTS I_Queue
VAR_INPUT
	ipList : I_List; // List to perform operations on.
END_VAR

METHOD PROTECTED NullReferenceException : BOOL
NullReferenceException := THIS^.ipList = 0;
IF NOT NullReferenceException THEN RETURN; END_IF
THIS^.RaiseException(2000+GVL_CmpErrors.ERR_INVALID_REFERENCE, 'Null or Invalid Reference');
END_METHOD

(* Number of items in queue*)
PROPERTY _Count : T_Capacity
GET
IF THIS^.NullReferenceException() THEN _Count := -1;RETURN; END_IF
_Count := THIS^.ipList._Count;
END_GET
END_PROPERTY

PROPERTY _Error_Status : ST_ERROR
GET
IF THIS^.NullReferenceException() THEN _Error_Status := THIS^.stError; RETURN; END_IF
THIS^.stError := THIS^.ipList._Error_Status;
_Error_Status := F_Error(THIS^.stError.bSTATUS, THIS^.stError.nCODE, THIS^.stError.sSOURCE);
END_GET
END_PROPERTY

(* Checks of queue is empty.*)
PROPERTY _Is_Empty : BOOL
GET
IF THIS^.NullReferenceException() THEN _Is_Empty := TRUE; RETURN; END_IF
_Is_Empty := THIS^.ipList._Is_Empty;
END_GET
END_PROPERTY

METHOD PROTECTED CatchError : BOOL
VAR_INPUT
END_VAR
IF THIS^.NullReferenceException() THEN RETURN; END_IF
THIS^.stError := ipList._Error_Status;
CatchError := stError.bSTATUS;
END_METHOD

